// TIA Portal V16 program export: 2 tag tables, 2 data types, 2 data blocks, 72 code blocks (in call order from the OBs), 28 instance data blocks

VAR_GLOBAL   // PLC tag table "Стандартная таблица переменных"
   "K1-112 2L1" AT %I0.0 : Bool;   // Реле безопастности К10 ОСНОВНАЯ напряжение управления
   "K1-113/1 3L1" AT %I0.1 : Bool;   // Реле безопастности К11 концевики группа 211,212,213,214
   "K1-113/2 4L1" AT %I0.2 : Bool;   // Реле безопастности К21 группа 221,222,224,225,231-235,311,312,313-317
   "K1-113/3 5L1" AT %I0.3 : Bool;   // Релле безопасности К31 группа 321,322,324
   "k1-113/4 6L1" AT %I0.4 : Bool;   // Релле безопасности К41 группа 331,332-337
   Varalla AT %I0.5 : Bool;   // резерв
   Varalla1 AT %I0.6 : Bool;   // резерв
   Varalla2 AT %I0.7 : Bool;   // резерв
   "211K1/211K2" AT %I1.0 : Bool;   // М211 включен сигналы
   "212K1" AT %I1.1 : Bool;   // Контактор К1 Включен М212 сигналы
   "213K1" AT %I1.2 : Bool;   // контактор К1 Включен М213 сигналы
   "311K1/311K2" AT %I1.3 : Bool;   // М311 включен сигналы
   Varalla3 AT %I1.4 : Bool;   // резерв
   Varalla4 AT %I1.5 : Bool;   // резерв
   Varalla5 AT %I1.6 : Bool;   // резерв
   Varalla6 AT %I1.7 : Bool;   // резерв
   "221K1" AT %I2.0 : Bool;   // М221 включен сигналы
   "222K1" AT %I2.1 : Bool;   // Контактор К1 Включен М222 сигналы
   "223K1" AT %I2.2 : Bool;   // Обратная связь
   "224K1" AT %I2.3 : Bool;   // М224 включен сигналы
   "225K1" AT %I2.4 : Bool;   // Контактор К1 Включен М225 сигналы
   "330K1" AT %I2.5 : Bool;   // Контактор К1 Включен М330 сигнал
   Varalla8 AT %I2.6 : Bool;   // резерв
   Varalla9 AT %I2.7 : Bool;   // резерв
   "231K1" AT %I3.0 : Bool;   // Контактор К1 Включен М231 сигналы
   "232K1" AT %I3.1 : Bool;   // Контактор К1- Включен М232 сигналы
   "233K1" AT %I3.2 : Bool;   // Контактор К1- Включен М233 сигналы
   "234K1" AT %I3.3 : Bool;   // М234 включен сигналы
   "235K1/235K2" AT %I3.4 : Bool;   // М235 включен сигналы
   Varalla10 AT %I3.5 : Bool;   // резерв
   Varalla11 AT %I3.6 : Bool;   // резерв
   Varalla12 AT %I3.7 : Bool;   // резерв
   "214K1" AT %I4.0 : Bool;   // М214 включен сигналы
   "312K1" AT %I4.1 : Bool;   // М312 включен сигналы
   "313K1/313K2" AT %I4.2 : Bool;   // М313 включен сигналы
   "314K1" AT %I4.3 : Bool;   // М314 включен сигналы
   "315K1" AT %I4.4 : Bool;   // М315 включен сигналы
   "316K1" AT %I4.5 : Bool;   // М316 включен сигналы
   "317K1" AT %I4.6 : Bool;   // Контактор К1 включен М317 сигналы
   Varalla13 AT %I4.7 : Bool;   // резерв
   "321K1/321K2" AT %I5.0 : Bool;   // М321 включен сигналы
   "322K1/322K2" AT %I5.1 : Bool;   // М322 включен сигналы
   "323K1/323K2" AT %I5.2 : Bool;   // М323 включен сигнал
   "K1-324U.1" AT %I5.3 : Bool;   // ПЧТ 324 в работе сигналы
   "325K1" AT %I5.4 : Bool;   // Контактор К1 М325 сигнал
   Varalla15 AT %I5.5 : Bool;   // резерв
   Varalla16 AT %I5.6 : Bool;   // резеов
   Varalla17 AT %I5.7 : Bool;   // резерв
   "331K1" AT %I6.0 : Bool;   // М331 включен сигналы
   "332K1" AT %I6.1 : Bool;   // Контактор К1- включен М332 сигналы
   "333K1" AT %I6.2 : Bool;   // Контактор К1 -включен М333 сигналы
   "334K1" AT %I6.3 : Bool;   // Контактор К1- включен М334 сигналы
   "335K1" AT %I6.4 : Bool;   // Контактор К1- включен М335 сигналы
   "336K1" AT %I6.5 : Bool;   // Контактор К1- включен М336 сигналы
   "337K1" AT %I6.6 : Bool;   // Контактор К1-включен М337 сигнал
   "K1-323U1" AT %I6.7 : Bool;   // ПЧТ 312 в работе сигналы
   "K1-212U1" AT %I7.0 : Bool;   // ПЧТ 212 в работе сигналы
   "K1-213U1" AT %I7.1 : Bool;   // ПЧТ 213 в работе сигналы
   "K1-215U1" AT %I7.2 : Bool;   // ПЧТ 215 в работе сигналы
   "K1-222U1" AT %I7.3 : Bool;   // ПЧТ 222 в работе сигналы
   "K1-225U1" AT %I7.4 : Bool;   // Пчт 225 в работе сигналы
   "K1-231U1" AT %I7.5 : Bool;   // ПЧТ 231 в работе сигналы
   "K1-233U1" AT %I7.6 : Bool;   // ПЧТ 233 в работе сигналы
   "K1-317U1" AT %I7.7 : Bool;   // ПЧТ 317 в работе сигналы
   "K1-332U1" AT %I8.0 : Bool;   // ПЧТ 332 в работе сигналы
   "K1-333U1" AT %I8.1 : Bool;   // ПЧТ 333 в работе сигналы
   "K1-334U1" AT %I8.2 : Bool;   // ПЧТ 334 в работе сигналы
   "K1-335U1" AT %I8.3 : Bool;   // ПЧТ 335 в работе сигналы
   "K1-336U1" AT %I8.4 : Bool;   // ПЧТ 336 в работе сигналы
   "K1-223U1" AT %I8.5 : Bool;   // ПЧТ М223 в работе сигнал
   "K1-324U1" AT %I8.6 : Bool;   // ПЧТ М324 в работе сигнал
   "K1-325U1" AT %I8.7 : Bool;   // ПЧТ М325 в работе сигнал
   "K1/112-S1" AT %I9.0 : Bool;   // Состояние концевика 112S1 сигналы
   "K1/112-S2" AT %I9.1 : Bool;   // Состояние концевика 112S2 сигналы
   "K1/112-S3" AT %I9.2 : Bool;   // Состояние концевика 112S3 сигналы
   Varalla22 AT %I9.3 : Bool;   // резерв
   "K1/113-S11" AT %I9.4 : Bool;   // Состояние концевиков 113S11 сигналы
   "K1/113-S12" AT %I9.5 : Bool;   // Состояние концевиков 113S12 сигналы
   "k1/113-S13" AT %I9.6 : Bool;   // Состояние концевиков 113S13 сигналы
   "FC 323.1" AT %I9.7 : Bool;   // Датчик блокировки поштучной
   "FC 323.2" AT %I10.0 : Bool;   // Датчик на останов основной горки
   "FC 223.1" AT %I10.1 : Bool;   // Начало зоны оценки
   "FC 223.2" AT %I10.2 : Bool;   // Конец зоны оценки
   "FC 223.3" AT %I10.3 : Bool;   // Сброс доски в брак
   FC_323_1 AT %I10.4 : Bool;   // резерв
   Key_Faser AT %I10.5 : Bool;   // индуктивник положения поштучной выдачи
   Varalla30 AT %I10.6 : Bool;   // резерв
   Varalla31 AT %I10.7 : Bool;   // резерв
   "Lift Upp" AT %I11.0 : Bool;   // Лифт вниз
   "Lift Down" AT %I11.1 : Bool;   // Лифт в верх
   "sloi doski" AT %I11.2 : Bool;   // Слой доски 1
   "sloi doski2" AT %I11.3 : Bool;   // Слой доски 2
   "doska v priymke elevator" AT %I11.4 : Bool;   // Доска в приямке элеватора
   koncevik1 AT %I11.5 : Bool;   // концевик 1(середина приемного транспортера)
   koncevik2 AT %I11.6 : Bool;   // концевик 2 (вилы лифта приемного транспортера)
   "nakloniy transporter" AT %I11.7 : Bool;   // наклонный транспортер датчик
   "1,8m" AT %I12.0 : Bool;   // 1,8 длинна
   "2,1m" AT %I12.1 : Bool;   // 2,1 длинна
   "2,4m" AT %I12.2 : Bool;   // 2,4 длинна
   "2,7m" AT %I12.3 : Bool;   // 2,7 длинна
   "3,0m" AT %I12.4 : Bool;   // 3,0 длинна
   "3,3m" AT %I12.5 : Bool;   // 3,3 длинна
   "3,6m" AT %I12.6 : Bool;   // 3,6 длинна
   "3,9m" AT %I12.7 : Bool;   // 3,9 длинна
   "4,2m" AT %I13.0 : Bool;   // 4,2 длинна
   "4,5m" AT %I13.1 : Bool;   // 4,5 длинна
   "4,8m" AT %I13.2 : Bool;   // 4,8 длинна
   "5,1m" AT %I13.3 : Bool;   // 5,1 длинна
   "5,4m" AT %I13.4 : Bool;   // 5,4 длинна
   "5,7m" AT %I13.5 : Bool;   // 5,7 длинна
   "6,0m" AT %I13.6 : Bool;   // 6,0 длинна
   PodBort_1 AT %I13.7 : Bool;   // Положение подвижного борта_1
   PodBort_2 AT %I14.0 : Bool;   // Положение подвижного борта _2
   K312Fault AT %I14.1 : Bool;   // Авария частотника 312
   "S14.2" AT %I14.2 : Bool;   // Максимальная ширина доски концевик М225 зона
   "S14.3" AT %I14.3 : Bool;   // Минимальная ширина доски концевик М225 зона
   "B14.4" AT %I14.4 : Bool;   // счет доски М225 зона после бобышек
   "B14.5" AT %I14.5 : Bool;   // счет доски М225 зона после бобышек
   "K-312U1" AT %I14.6 : Bool;   // ПЧТ 312 В работе
   "S14.7" AT %I14.7 : Bool;   // заднее положение вил
   "S15.0" AT %I15.0 : Bool;   // замедление вил назад
   "S15.1" AT %I15.1 : Bool;   // замедление в перед вил
   "S15.2" AT %I15.2 : Bool;   // Переднее положение вил
   "311_S1" AT %I15.3 : Bool;   // Запрет двиджения М311
   Index AT %I15.4 : Bool;   // Индексная точка энкодера
   "B15.5" AT %I15.5 : Bool;   // вилы в верху
   "311_S2" AT %I15.6 : Bool;   // Ручное управление М311
   "B15.7" AT %I15.7 : Bool;   // вилы в низу
   FC_232_1 AT %I16.0 : Bool;   // набор слоя пакета на лифте1
   "S16.1" AT %I16.1 : Bool;   // лифт ПфМ в низу
   "S16.2" AT %I16.2 : Bool;   // лифт ПФМ в верху
   FC_225_Upor AT %I16.3 : Bool;   // датчик доски на упорах перед транспортером с бобышками
   "E16.4" AT %I16.4 : Bool;   // Уровень Гидростанции Основной
   FC_232_2 AT %I16.5 : Bool;   // Набор слоя пакета на лифте2
   KeyFazerPFM_repeater AT %I16.6 : Bool;   // Второй кейфазер на транспортер бобышек
   KeyFazerPFM AT %I16.7 : Bool;   // кейфазер для транспортера бобышек
   "B17.0" AT %I17.0 : Bool;   // наличие прокладок на М312
   "B17.1" AT %I17.1 : Bool;   // наличие прокладки в М314
   "B17.2" AT %I17.2 : Bool;   // наличие прокладки в М315
   "234.4" AT %I17.3 : Bool;   // второй датчик наличия прокладки перед каруселью
   "234.1" AT %I17.4 : Bool;   // 234.1 прокладка на выдаче(датчик)
   "234.2" AT %I17.5 : Bool;   // 234.2 прокладка максимальный слой
   "234.3" AT %I17.6 : Bool;   // 234.3 перекос прокладки (Авария)
   Fc316 AT %I17.7 : Bool;   // Датчик в конце М316 перед элеватором1
   "B18.0" AT %I18.0 : Bool;   // рейкоукладчик в верху
   "B18.1" AT %I18.1 : Bool;   // второй индуктив на позиционирование карусели
   "S18.2" AT %I18.2 : Bool;   // среднее положение рейкоукладчика
   "S18.3" AT %I18.3 : Bool;   // рейкоукладчик в низу
   "B18.4" AT %I18.4 : Bool;   // датчик положения захвата прокладки открыто
   "B18.5" AT %I18.5 : Bool;   // датчик положени захвата прокладки закрыто
   "B18.6" AT %I18.6 : Bool;   // сигнал набора слоя
   "B18.7" AT %I18.7 : Bool;   // Остановка транспортера прокладок
   "B19.0" AT %I19.0 : Bool;   // Обратный ход транспортера прокладок ДАТЧИК
   Varalla35 AT %I19.1 : Bool;   // резерв
   Varalla36 AT %I19.2 : Bool;   // резерв
   Varalla37 AT %I19.3 : Bool;   // резерв
   Varalla38 AT %I19.4 : Bool;   // резерв
   Varalla39 AT %I19.5 : Bool;   // резерв
   Varalla40 AT %I19.6 : Bool;   // резерв
   Varalla41 AT %I19.7 : Bool;   // резерв
   Varalla42 AT %I20.0 : Bool;   // резерв
   Varalla43 AT %I20.1 : Bool;   // резерв
   Varalla44 AT %I20.2 : Bool;   // резерв
   Varalla45 AT %I20.3 : Bool;   // резерв
   Varalla46 AT %I20.4 : Bool;   // резерв
   Varalla47 AT %I20.5 : Bool;   // резерв
   Varalla48 AT %I20.6 : Bool;   // резерв
   Varalla49 AT %I20.7 : Bool;   // резерв
   Varalla50 AT %I21.0 : Bool;   // резерв
   Varalla51 AT %I21.1 : Bool;   // резерв
   Varalla52 AT %I21.2 : Bool;   // резерв
   Varalla53 AT %I21.3 : Bool;   // резерв
   Varalla54 AT %I21.4 : Bool;   // резерв
   Varalla55 AT %I21.5 : Bool;   // резерв
   Varalla56 AT %I21.6 : Bool;   // резерв
   Varalla57 AT %I21.7 : Bool;   // резерв
   "B22.0" AT %I22.0 : Bool;   // доска в конце роликового транспортера(брак)
   "B22.1" AT %I22.1 : Bool;   // доска в начале роликового транспортера(брак)
   "S22.2" AT %I22.2 : Bool;   // вилы брака ПФМ в перед
   "S22.3" AT %I22.3 : Bool;   // вилы брака ПФМ назад
   "B22.4" AT %I22.4 : Bool;   // лифт брака ПФМ в верху
   "B22.5" AT %I22.5 : Bool;   // лифт брака ПФМ в низу
   "B22.6" AT %I22.6 : Bool;   // Слой на вилах брака ПФМ
   "FC 22.7" AT %I22.7 : Bool;   // Счет доски слоя на пфм Брака
   "B23.0" AT %I23.0 : Bool;   // Пакет на основном разгрузочном транспортере3
   "B23.1" AT %I23.1 : Bool;   // пакет на разгрузочном транспортере 2
   M324Sync AT %I23.2 : Bool;   // индуктив синхронизации М 324
   Varalla60 AT %I23.3 : Bool;   // резерв
   Varalla61 AT %I23.4 : Bool;   // резерв
   Varalla62 AT %I23.5 : Bool;   // резерв
   "FC 23.6" AT %I23.6 : Bool;   // Упоры подняты ПФМ брака
   "FC 23.7" AT %I23.7 : Bool;   // Упоры опущены ПФМ брака
   S76 AT %I24.0 : Bool;   // стоповая кнопка OP1
   "S76.1" AT %I24.1 : Bool;   // Включение напряжения управления
   "S76.2" AT %I24.2 : Bool;   // Подтверждение ошибки
   "S76.3" AT %I24.3 : Bool;   // Гидравлика линии в положении включено
   "E76.4" AT %I24.4 : Bool;   // Старт гидравлики
   "S76.5" AT %I24.5 : Bool;   // авто включение и выключение загрузчика ( режим авто всей загрузки)
   "S76.6" AT %I24.6 : Bool;   // авто М211 приемный транспортер
   "E76.7" AT %I24.7 : Bool;   // вперед М211 приемный транспортер в автомате
   "S77.0" AT %I25.0 : Bool;   // авто М222 горка
   "E77.1" AT %I25.1 : Bool;   // вперед М222 горка в автомате
   "S77.2" AT %I25.2 : Bool;   // Квитирование зоны 1(от горки до ПФМ)
   "S77.3" AT %I25.3 : Bool;   // Квитирование зоны выгрузки
   "S77.4" AT %I25.4 : Bool;   // Квитирование зоны 2 (ПФМ брака)
   "S77.5" AT %I25.5 : Bool;   // авто режим зоны 1( включено, выключено) ( от горки до ПФМ)
   "S77.6" AT %I25.6 : Bool;   // Выдвинуть упоры поштучника
   "E77.7" AT %I25.7 : Bool;   // Убрать упоры поштучника
   "S78.0" AT %I26.0 : Bool;   // Вилы выдвинуть
   "E78.1" AT %I26.1 : Bool;   // Вилы задвинуть
   "S78.2" AT %I26.2 : Bool;   // Вилы опустить
   "E78.3" AT %I26.3 : Bool;   // Вилы поднять
   "S78.4" AT %I26.4 : Bool;   // Лифт опустить
   "E78.5" AT %I26.5 : Bool;   // Лифт поднять
   "S78.6" AT %I26.6 : Bool;   // рейкоукладчик вниз
   "E78.7" AT %I26.7 : Bool;   // рейкоукладчик вверх
   "S79.0" AT %I27.0 : Bool;   // принудительно завершить сборку пакета
   "S79.1" AT %I27.1 : Bool;   // авто подача прокладки(включен,выключен)
   "E79.2" AT %I27.2 : Bool;   // резерв
   "S79.3" AT %I27.3 : Bool;   // авто режим ПФМ брака (включено,выключено)
   "S79.4" AT %I27.4 : Bool;   // Сброс с рольганга(брака) вперпед
   "S79.5" AT %I27.5 : Bool;   // Транспортер набора слоя ( брака) вперед
   "S79.6" AT %I27.6 : Bool;   // вилы( брака) вперед
   "E79.7" AT %I27.7 : Bool;   // вилы( брака) назад
   "S80.0" AT %I28.0 : Bool;   // Упоры слоя ПФМ( брака)
   "E80.1" AT %I28.1 : Bool;   // Упоры слоя ПФМ( брака)
   "S80.2" AT %I28.2 : Bool;   // Лифт ПФМ(брака) опустить
   "E80.3" AT %I28.3 : Bool;   // Лифт ПФМ(брака) поднять
   "S80.4" AT %I28.4 : Bool;   // поднять, опустить Подвижный борт(М235)
   "S80.5" AT %I28.5 : Bool;   // вперед подвижный борт(М235)
   "E80.6" AT %I28.6 : Bool;   // назад подвижный борт(М235)
   "S80.7" AT %I28.7 : Bool;
   Varalla106 AT %I29.0 : Bool;   // резерв
   Varalla107 AT %I29.1 : Bool;   // резерв
   Varalla108 AT %I29.2 : Bool;   // резерв
   Varalla109 AT %I29.3 : Bool;   // резерв
   Varalla110 AT %I29.4 : Bool;   // резерв
   Varalla111 AT %I29.5 : Bool;   // резерв
   Varalla112 AT %I29.6 : Bool;   // резерв
   Varalla113 AT %I29.7 : Bool;   // резерв
   "S82.0" AT %I30.0 : Bool;   // Стоп ОР2
   "S81.1" AT %I30.1 : Bool;   // Приемный транспортер вперед ОР2
   "E82.2" AT %I30.2 : Bool;   // Приемный транспортер назад ОР2
   "S82.3" AT %I30.3 : Bool;   // Авто загрузка включена,выключена ОР2
   "S82.4" AT %I30.4 : Bool;   // Лифт загрузки поднять ОР2
   "E82.5" AT %I30.5 : Bool;   // Лифт загрузки опустить ОР2
   "S82.6" AT %I30.6 : Bool;   // Наклонный транспортер авто ОР2
   "E82.7" AT %I30.7 : Bool;   // Авто наклонный транспортер вперед ОР2
   "S83.0" AT %I31.0 : Bool;   // Ленточный транспортер удаления прокладок назад ОР2
   "E83.1" AT %I31.1 : Bool;   // Ленточный транспортер удаления прокладок вперед ОР2
   "E83.2" AT %I31.2 : Bool;   // Горка прокладок 1 авто ОР2
   "E83.3" AT %I31.3 : Bool;   // Горка прокладок 1 вперед ОР2(авто)
   "S83.4" AT %I31.4 : Bool;   // Квитирование зоны 1 ОР2
   Varalla114 AT %I31.5 : Bool;   // резерв
   Varalla115 AT %I31.6 : Bool;   // резерв
   Varalla116 AT %I31.7 : Bool;   // резерв
   "S84.0" AT %I32.0 : Bool;   // Стоп ОР3
   "S84.1" AT %I32.1 : Bool;   // Транспортер М317 прокладок вперед ОР3
   "E84.2" AT %I32.2 : Bool;   // Транспортер М317 прокладок назад ОР3
   "S84.3" AT %I32.3 : Bool;   // Дозированиe включено ОР3
   "S84.4" AT %I32.4 : Bool;   // авто подача прокладок включена, выключена ОР3
   "S84.5" AT %I32.5 : Bool;   // Рейкоукладчик вниз ОР3
   "E84.6" AT %I32.6 : Bool;   // Рейкоукладчик вверх ОР3
   "S84.7" AT %I32.7 : Bool;   // Открыть стакан прокладки ОР3
   "E85.0" AT %I33.0 : Bool;   // Закрыть стакан прокладки ОР3
   "S85.1" AT %I33.1 : Bool;
   "E85.2" AT %I33.2 : Bool;
   "S85.3" AT %I33.3 : Bool;   // авто горка прокладок 2,3 ОР3
   "E85.4" AT %I33.4 : Bool;   // горка 2,3 прокладок вперед(авто) ОР3
   "S85.5" AT %I33.5 : Bool;   // М234 назад ОР3
   "E85.6" AT %I33.6 : Bool;   // М234 вперед транспортер прокладок перед крючками ОР3
   "S85.7" AT %I33.7 : Bool;   // Квитирование зоны прокладок ОР3
   "S86.0" AT %I34.0 : Bool;   // Лифт ПФМ вниз ОР3
   "E86.1" AT %I34.1 : Bool;   // ЛИфт ПФМ вверх ОР3
   "S86.2" AT %I34.2 : Bool;   // Ролики лифта ПФМ вперед ОР3
   "S86.3" AT %I34.3 : Bool;   // ПФМ Основное Авто включено, выключено ОР3
   "S86.4" AT %I34.4 : Bool;   // Подтверждение неисправности ОР3
   "S86.5" AT %I34.5 : Bool;   // датчик
   Varalla117 AT %I34.6 : Bool;   // резерв
   Varalla118 AT %I34.7 : Bool;   // резерв
   "S87.0" AT %I35.0 : Bool;   // Кнопка брака ОР1.1
   "S87.1" AT %I35.1 : Bool;   // Горка авто ОР1.1
   "E87.2" AT %I35.2 : Bool;   // Горка ОР1.1 (авто)
   "S87.3" AT %I35.3 : Bool;   // датчик перекоса перед плавниками
   "S87.4" AT %I35.4 : Bool;   // набор ковра перед плавниками
   Varalla119 AT %I35.5 : Bool;   // резерв
   Varalla120 AT %I35.6 : Bool;   // резерв
   Varalla121 AT %I35.7 : Bool;   // резерв
   "S88.0" AT %I36.0 : Bool;   // Стоп ОР4
   "K3.3" AT %I36.1 : Bool;   // работа подвижного борта ОР4
   "S88.2" AT %I36.2 : Bool;   // Выкатной транспортер 1 ПФМ назад ОР4
   "E88.3" AT %I36.3 : Bool;   // Выкатной транспортер 1 ПФМ вперед ОР4
   "S88.4" AT %I36.4 : Bool;   // Выкатной транспортер 2 ПФМ назад ОР4
   "S88.5" AT %I36.5 : Bool;   // Выкатной транспортер 2 ПФМ вперед ОР4
   "E88.6" AT %I36.6 : Bool;   // резерв ОР4
   "S88.7" AT %I36.7 : Bool;   // резерв ОР4
   "S89.0" AT %I37.0 : Bool;   // Выкатной транспортер 3 ПФМ назад ОР4
   "S89.1" AT %I37.1 : Bool;   // Выкатной транспортер 3 ПФМ вперед ОР4
   "S89.2" AT %I37.2 : Bool;   // Квитирование ОР4
   "S89.3" AT %I37.3 : Bool;   // датчик ОР4
   Varalla122 AT %I37.4 : Bool;   // резерв ОР4
   Varalla123 AT %I37.5 : Bool;   // резерв ОР4
   Varalla124 AT %I37.6 : Bool;   // резерв ОР4
   Varalla125 AT %I37.7 : Bool;   // резерв ОР4
   "S90.0" AT %I38.0 : Bool;   // Стоп ОР5
   "S90.1" AT %I38.1 : Bool;   // М331 вперед ленточный транспортер брака ОР5
   "S90.2" AT %I38.2 : Bool;   // М332 вперед сбрасыватель рольганга брака ОР5
   Varalla126 AT %I38.3 : Bool;   // резерв
   "S90.4" AT %I38.4 : Bool;   // Вилы ПФМ брака назад ОР5
   "E90.5" AT %I38.5 : Bool;   // Вилы ПФМ брака вперед ОР5
   "S90.6" AT %I38.6 : Bool;   // Опустить упоры формирования слоя на ПФМ брака ОР5
   "E90.7" AT %I38.7 : Bool;   // Поднять упоры формирования слоя на ПФМ брака ОР5
   "S91.0" AT %I39.0 : Bool;   // Лифт брака ПФМ опустить ОР5
   "E91.1" AT %I39.1 : Bool;   // Лифт брака ПФМ поднять ОР5
   "S91.2" AT %I39.2 : Bool;   // квитирование ПФМ 2
   Varalla127 AT %I39.3 : Bool;   // резерв
   Varalla128 AT %I39.4 : Bool;   // резерв
   Varalla129 AT %I39.5 : Bool;   // резерв
   Varalla130 AT %I39.6 : Bool;   // резерв
   Varalla131 AT %I39.7 : Bool;   // резерв
   "K1-212U" AT %QW512 : Int;
   "K1-213U" AT %QW514 : Int;
   "K1-215U" AT %QW516 : Int;
   "K1-222U" AT %QW518 : Int;
   "K1-225U" AT %QW520 : Int;
   "K1-231U" AT %QW522 : Int;
   "K1-233U" AT %QW524 : Int;
   "K1-317U" AT %QW526 : Int;
   "K1-332U" AT %QW528 : Int;
   "K1-333U" AT %QW530 : Int;
   "K1-334U" AT %QW532 : Int;
   "K1-335U" AT %QW534 : Int;
   "K1-336U" AT %QW536 : Int;
   "K1-223U" AT %QW538 : Int;
   "k1-323U" AT %QW540 : Int;
   "K1-325U" AT %QW542 : Int;
   "K1-112x1" AT %Q0.0 : Bool;   // релле Сирены
   "Sk1-113" AT %Q0.1 : Bool;   // разрешение на запуск релле К10 безопастность
   "K1-113X1" AT %Q0.2 : Bool;   // разрешение на запуск релле К11 безопастность
   "K1-113X2" AT %Q0.3 : Bool;   // разрешение на запуск релле К21 безопастность
   "K1-113X3" AT %Q0.4 : Bool;   // разрешение на запуск релле К31 безопастность
   "K1-113X4" AT %Q0.5 : Bool;   // разрешение на запуск релле К41 безопастность
   Varalla65 AT %Q0.6 : Bool;   // резерв
   Varalla66 AT %Q0.7 : Bool;   // резерв
   "K1-211X1" AT %Q1.0 : Bool;   // М211 вперед загрузочный транспортер
   "K1-211X1.1" AT %Q1.1 : Bool;   // М211 назад загрузочный транспортер
   "K1-212X1" AT %Q1.2 : Bool;   // контактор К1-212 ПЧТ запуск лифт
   "K1-212X1.1" AT %Q1.3 : Bool;   // Растормаживание М212 лифт
   "K1-213X1" AT %Q1.4 : Bool;   // контактор К1-213 ПЧТ запуск наклонный транспортер
   "K1-311X1" AT %Q1.5 : Bool;   // запуск ленточного транспортера удалителя прокладок M311
   Varalla68 AT %Q1.6 : Bool;   // резерв
   Varralla69 AT %Q1.7 : Bool;   // резерв
   "K1-221X1" AT %Q2.0 : Bool;   // запуск М221 гидростанция1
   "K1-222X1" AT %Q2.1 : Bool;   // Запуск контактора К1-222 ПЧТ основной элеватор
   "K1-223X1" AT %Q2.2 : Bool;   // запуск М223 Цепной после поштучника
   "K1-224X1" AT %Q2.3 : Bool;   // запуск М224 выдвинуть упоры поштучника
   "K1-224-x1.1" AT %Q2.4 : Bool;   // запуск М224 задвинуть упоры поштучника
   "K1-225X1" AT %Q2.5 : Bool;   // включение контактора К1-225 ПЧТ транспортер бобышек
   "K1-231X1" AT %Q2.6 : Bool;   // включение контактора К1-231 ПЧТ ролики торцовочные
   "K1-232X1" AT %Q2.7 : Bool;   // включение контактора К1-232 ПЧТ Лифт ПФМ
   "K1-232X1.1" AT %Q3.0 : Bool;   // Тормоз Лифта ПФМ
   "K1-233X1" AT %Q3.1 : Bool;   // включение контактора К1-233 ПЧТ вилы ПФМ
   "K1-234X1" AT %Q3.2 : Bool;   // запуск М234 транспортер прокладок перед крючками ПФМ
   "K1-235X1" AT %Q3.3 : Bool;   // запуск М235 вперед подвижный борт
   "K1-214X1" AT %Q3.4 : Bool;   // запуск М214 транспортер загрузки прокладок
   "K1-330X1" AT %Q3.5 : Bool;   // запуск М330 контактора лента брака2
   "K1-312X1" AT %Q3.6 : Bool;   // запуск М312 первая горка прокладок
   "K1-313X1" AT %Q3.7 : Bool;   // запуск М313 вперед транспортер прокладок после первой горки
   "K1-313X1.1" AT %Q4.0 : Bool;   // запуск М313 назад транспортера прокладок после первой горки
   "K1-314X1" AT %Q4.1 : Bool;   // запуск М314 горка прокладок 2
   "K1-315X1" AT %Q4.2 : Bool;   // запуск М315 горка прокладок 3
   "K1-316X1" AT %Q4.3 : Bool;   // запуск М316 транспортер загрузки прокладок в горку 2
   "K1-317X1" AT %Q4.4 : Bool;   // включение контактора К1-317 ПЧТ основной транспортер прокладок
   "K1-317X1.1" AT %Q4.5 : Bool;   // тормоз М317
   "K1-321X1" AT %Q4.6 : Bool;   // запуск М321 вперед выкатной транспортер ПФМ
   "K1-321X1.1" AT %Q4.7 : Bool;   // запуск М321 назад выкатной транспортер ПФМ
   "K1-322X1" AT %Q5.0 : Bool;   // запуск М322 вперед выкатной транспортер ПФМ2
   "K1-322X1.1" AT %Q5.1 : Bool;   // Запуск М322 назад выкатной транспортер ПФМ2
   "K1-323X1" AT %Q5.2 : Bool;   // Запуск контактора М323 маленький после элеватора
   "K1-325U2" AT %Q5.3 : Bool;   // Старт ПЧТ М325 набор слоя основной
   "K1-324U2" AT %Q5.4 : Bool;   // команда на ПЧТ вперед М324 выгрузка покета выкатной ПФМ3
   "K1-324U2.2" AT %Q5.5 : Bool;   // команда на ПЧТ назад М324 выгрузка покета выкатной ПФМ3
   "K1-325X1" AT %Q5.6 : Bool;   // Включение контактора К1-325 ПЧТ набор слоя основной
   "K1-235X1.1" AT %Q5.7 : Bool;   // запуск М235 назад подвижный борт
   "K1-331X1" AT %Q6.0 : Bool;   // запуск М331 ленточный транспортер брака
   "K1-332x1" AT %Q6.1 : Bool;   // включение контактора К1-332 ПЧТ сбрасыватель с рольганга (брак)
   "K1--333X1" AT %Q6.2 : Bool;   // включение контактора К1-333 ПЧТ рольганг (брака)
   "K1-334X1" AT %Q6.3 : Bool;   // включение контактора К1-334 ПЧТ транспортер сбора слоя ПФМ брака
   "K1-335X1" AT %Q6.4 : Bool;   // включение контактора К1-335 ПЧТ вилы ПФМ брака
   "K1-336X1" AT %Q6.5 : Bool;   // Включение контактора К1-336 ПЧТ лифт ПФМ брака
   "K1-336X1.1" AT %Q6.6 : Bool;   // Тормоз М336 лифта ПФМ брака
   "K1-337K1" AT %Q6.7 : Bool;   // Контактор пуска Гирдростанции ПФМ Брака
   Varalla70 AT %Q7.0 : Bool;   // резерв
   "K1-312U2" AT %Q7.1 : Bool;   // Старт ПЧТ 312
   Varalla72 AT %Q7.2 : Bool;   // резерв
   Varalla73 AT %Q7.3 : Bool;   // резерв
   Varalla74 AT %Q7.4 : Bool;   // резерв
   Varalla75 AT %Q7.5 : Bool;   // резерв
   Varalla76 AT %Q7.6 : Bool;   // резерв
   Varalla77 AT %Q7.7 : Bool;   // резерв
   "K1-212U2" AT %Q8.0 : Bool;   // старт ПЧТ М212
   "K1-212U2.2" AT %Q8.1 : Bool;   // Реверс ПЧТ М212
   "K1-213U2" AT %Q8.2 : Bool;   // Старт ПЧТ М213
   "K1-215U2" AT %Q8.3 : Bool;   // Старт ПЧТ 232
   "K1-215U2.2" AT %Q8.4 : Bool;   // Реверс ПЧТ 232
   "K1-222U2" AT %Q8.5 : Bool;   // Старт ПЧТ 222
   "K1-225U2" AT %Q8.6 : Bool;   // Старт ПЧТ 225
   "K1-231U2" AT %Q8.7 : Bool;   // Старт ПЧТ 231
   "K1-233U2" AT %Q9.0 : Bool;   // Старт ПЧТ 233
   "K1-233U2.2" AT %Q9.1 : Bool;   // Реверс ПЧТ 233
   "K1-223U2" AT %Q9.2 : Bool;   // Старт ПЧТ 223
   "K1-332U2" AT %Q9.3 : Bool;   // Старт ПЧТ 332
   "K1-333U2" AT %Q9.4 : Bool;   // Старт ПЧТ 333
   "K1-334U2" AT %Q9.5 : Bool;   // Старт ПЧТ 334
   "K1-335U2" AT %Q9.6 : Bool;   // Старт ПЧТ 335
   "K1-335U2.2" AT %Q9.7 : Bool;   // Реверс ПЧТ 335
   "K1-336U2" AT %Q10.0 : Bool;   // Стасрт ПЧТ 336
   "K1-336U2.2" AT %Q10.1 : Bool;   // Реверс ПЧТ 336
   "K1-317U2" AT %Q10.2 : Bool;   // Старт ПЧТ 317
   "K1-317U2.2" AT %Q10.3 : Bool;   // Реверс ПЧТ 317
   Y223_1 AT %Q12.0 : Bool;   // переворот доски вверх
   Y223_2 AT %Q12.1 : Bool;   // переворот доски вниз
   Y223_3 AT %Q12.2 : Bool;   // сброс в брак вниз
   Y223_4 AT %Q12.3 : Bool;   // сброс в брак вверх
   Y323_1 AT %Q12.4 : Bool;   // упоры перед поштучкой вверх
   Y323_2 AT %Q12.5 : Bool;   // упоры перед поштучкой вниз
   Upor_brak_up AT %Q12.6 : Bool;   // упоры ПФМ брака вверх
   Upor_brak_down AT %Q12.7 : Bool;   // упоры ПФМ брака вниз
   "Y223.3" AT %Q13.0 : Bool;   // перепускной клапан маленькая гидростанция
   "Y223.4" AT %Q13.1 : Bool;   // перепускной клапан маленькая гидростанция
   Varalla89 AT %Q11.6 : Bool;   // резерв
   Varalla90 AT %Q11.7 : Bool;   // резерв
   "K1-323U2" AT %Q10.4 : Bool;   // Старт ПЧТ 323
   "Y12.1" AT %Q10.5 : Bool;   // резерв
   Varalla91 AT %Q10.6 : Bool;   // резерв
   Varalla92 AT %Q10.7 : Bool;   // резерв
   Varalla93 AT %Q11.0 : Bool;   // резерв
   Varalla94 AT %Q11.1 : Bool;   // резерв
   Varalla95 AT %Q11.2 : Bool;   // резерв
   Varalla96 AT %Q11.3 : Bool;   // резерв
   "Y13.0" AT %Q11.4 : Bool;
   "Y13.1" AT %Q11.5 : Bool;
   "Y13.2" AT %Q13.2 : Bool;
   "Y13.3" AT %Q13.3 : Bool;
   "Y13.4" AT %Q13.4 : Bool;
   "Y13.5" AT %Q13.5 : Bool;
   "Y13.6" AT %Q13.6 : Bool;
   "Y13.7" AT %Q13.7 : Bool;
   Line1_1 AT %Q14.0 : Bool;   // вилы вниз
   Line1_2 AT %Q14.1 : Bool;   // вилы вверх
   Line2_1 AT %Q14.2 : Bool;   // упоры перед поштучкой вверх
   Line2_2 AT %Q14.3 : Bool;   // упоры перед поштучкой вниз
   Line3_1 AT %Q14.4 : Bool;   // подвижный борт опустить
   Line3_2 AT %Q14.5 : Bool;   // подвижный борт поднять
   Line4_1 AT %Q14.6 : Bool;   // выдача прокладки вниз
   Line4_2 AT %Q14.7 : Bool;   // выдача прокладки вверх
   Perepusk AT %Q15.0 : Bool;   // перепускной клапан большая гидростанция
   Line5_1 AT %Q15.1 : Bool;   // каретка прокладки вниз
   Line5_2 AT %Q15.2 : Bool;   // каретка прокладки вверх
   Line6_1 AT %Q15.3 : Bool;   // ложементы закрыть
   Line6_2 AT %Q15.4 : Bool;   // ложементы открыть
   Varalla100 AT %Q15.5 : Bool;   // резерв
   Varalla101 AT %Q15.6 : Bool;   // резерв
   Varalla102 AT %Q15.7 : Bool;   // резерв
   "H76.0" AT %Q16.0 : Bool;   // Напряжение управления включено (лампочка) ОР1
   "H76.1" AT %Q16.1 : Bool;   // потверждение аварии (лампочка) ОР1
   "H76.2" AT %Q16.2 : Bool;   // Гидравлика линии в положении включено (лампочка) ОР1
   "H76.3" AT %Q16.3 : Bool;   // авто включение и выключение загрузчика ( режим авто всей загрузки) (лампочка)ОР1
   "H76.4" AT %Q16.4 : Bool;   // разгрусчик открыт (лапмочка) ОР1
   "H76.5" AT %Q16.5 : Bool;   // Квитирование ПФМ 1 (лапмочка)ОР1
   "H76.6" AT %Q16.6 : Bool;   // Квитирование (лампочка)ОР1
   "H76.7" AT %Q16.7 : Bool;   // Квитирование ПФМ 2 (лампочка)ОР1
   "H77.0" AT %Q17.0 : Bool;   // ПФМ 1 авто включено ( лампочка)ОР1
   "H77.1" AT %Q17.1 : Bool;   // авто подача прокладки(включен,выключен) (лампочка)ОР1
   "H77.2" AT %Q17.2 : Bool;   // Авто ПФМ 2 включен (лампочка)ОР1
   Varalla132 AT %Q17.3 : Bool;   // резерв ОР1
   Varalla133 AT %Q17.4 : Bool;   // резерв ОР1
   Varalla134 AT %Q17.5 : Bool;   // резерв ОР1
   Varalla135 AT %Q17.6 : Bool;   // резерв ОР1
   Varalla136 AT %Q17.7 : Bool;   // резерв ОР1
   "H78.0" AT %Q18.0 : Bool;   // Авто загрузка включена,выключена ОР2 (лампочка)
   "H78.1" AT %Q18.1 : Bool;   // квитирование загрузки (лампочка)ОР2
   Varalla137 AT %Q18.2 : Bool;   // резерв
   Varalla138 AT %Q18.3 : Bool;   // резерв
   "A78.4" AT %Q18.4 : Bool;   // Авто подачи прокладок включен (лампочка)ОР3
   "A78.5" AT %Q18.5 : Bool;   // Квитирование прокладок (лампочка)ОР3
   "A78.6" AT %Q18.6 : Bool;   // Авто ПФМ 1 включен ( лампочка) ОР3
   "H78.7" AT %Q18.7 : Bool;   // Авария (лампочка)ОР3
   "H79.0" AT %Q19.0 : Bool;   // Квитирование выгрузки (лампочка) ОР4
   Pakkauspuristin AT %Q19.1 : Bool;
   "A79.2" AT %Q19.2 : Bool;   // резерв
   "A79.3" AT %Q19.3 : Bool;   // резерв
   "H79.4" AT %Q19.4 : Bool;   // Квитирование ПФМ2 (лампочка)
   Varalla139 AT %Q19.5 : Bool;   // резерв
   Varalla140 AT %Q19.6 : Bool;   // резерв
   Varalla141 AT %Q19.7 : Bool;   // резерв
   Lift AT %M20.0 : Bool;
   FALSE AT %M20.1 : Bool;
   M212StartDelay AT %T1 : Timer;   // Задержка перд стартом загрузки пакета на лифт
   Tag_2 AT %T2 : Timer;
   M212DownDelay AT %T3 : Timer;   // Задержка на опускания лифта вниз
   DropDelay AT %T4 : Timer;   // задержка на срабатывания датчиков сброся слоя
   m212waitAfterDrop AT %T6 : Timer;   // Задержка на сброс доски после сброса
   m213DropDelay AT %T7 : Timer;
   M212waitEmptyHole AT %T8 : Timer;   // Ожидание освобождения приямка горки загрузки
   Tag_9 AT %T9 : Timer;
   M211startDelay AT %T10 : Timer;   // задержка старта транспортера при установке пакета погрузчиком
   Tag_11 AT %T11 : Timer;
   Tag_12 AT %T12 : Timer;
   Tag_13 AT %T13 : Timer;
   Tag_14 AT %T14 : Timer;
   Tag_15 AT %T15 : Timer;
   Tag_16 AT %T16 : Timer;
   Tag_17 AT %T17 : Timer;
   Tag_18 AT %T18 : Timer;
   Tag_5 AT %M0.0 : Bool;
   Tag_61 AT %M0.1 : Bool;
   Tag_62 AT %T19 : Timer;
   NaprUpr AT %M0.6 : Bool;   // меркер напряжения управления
   Tag_19 AT %C1 : Counter;
   Tag_20 AT %C2 : Counter;
   HodVil2 AT %M1.2 : Bool;
   Tag_71 AT %T5 : Timer;
   Tag_72 AT %T20 : Timer;
   Tag_73 AT %C3 : Counter;
   Fouls AT %M4.0 : Bool;
   TRUE AT %M4.1 : Bool;
   "Tag_19(1)" AT %T21 : Timer;
   M213AlarmFilter AT %T22 : Timer;
   M214AlarmFilter AT %T23 : Timer;
   "221StartDelay" AT %T24 : Timer;
   "222AlarmFilter" AT %T25 : Timer;
   "223AlarmFilter" AT %T26 : Timer;
   "332AlarmFilter" AT %T27 : Timer;
   "333AlarmFilter" AT %T28 : Timer;
   "334AlarmFilter" AT %T29 : Timer;
   "336DownDelay" AT %T30 : Timer;
   "336AlarmFilter" AT %T31 : Timer;
   "321AlarmFilter" AT %T32 : Timer;
   "322AlarmFilter" AT %T33 : Timer;
   "324AlarmFilter" AT %T34 : Timer;
   "214AlarmFiltr" AT %T35 : Timer;
   "312AlarmFiltr" AT %T36 : Timer;
   "313AlarmFilter" AT %T37 : Timer;
   "316AlarmFiltr" AT %T38 : Timer;
   "314AlarmFilter" AT %T39 : Timer;
   "234AlarmFilter" AT %T40 : Timer;
   Tag_3 AT %M4.7 : Bool;
   "224AlarmFilter" AT %T41 : Timer;
   "225AlarmFilter" AT %T42 : Timer;
   "231AlarmFilter" AT %T43 : Timer;
   "235AlarmFilter" AT %T44 : Timer;
   "311AlarmFilter" AT %T45 : Timer;
   "335AlarmFilter" AT %T46 : Timer;
   "331AlarmFilter" AT %T47 : Timer;
   "233AlarmFilter" AT %T48 : Timer;
   "337AlarmFilter" AT %T49 : Timer;
   "232AlarmFilter" AT %T50 : Timer;
   alarm AT %M2.0 : Bool;
   M323_HoldRun AT %T51 : Timer;
   Tag_1 AT %C4 : Counter;
   Tag_4 AT %T52 : Timer;
   Tag_6 AT %M2.1 : Bool;
   M323_RunTask AT %T53 : Timer;
   Tag_7 AT %T54 : Timer;
   Tag_8 AT %T55 : Timer;
   ElevatorPFM_Defective_cmd_lowering AT %M4.5 : Bool;
   Tag_21 AT %T56 : Timer;
   Tag_22 AT %M40.0 : Bool;
   Tag_23 AT %M40.1 : Bool;
   Tag_24 AT %M40.2 : Bool;
   Tag_25 AT %M40.3 : Bool;
   Tag_26 AT %M40.4 : Bool;
   Tag_27 AT %M40.5 : Bool;
   Tag_28 AT %M40.6 : Bool;
   Tag_29 AT %M40.7 : Bool;
   Tag_30 AT %M41.0 : Bool;
   Tag_31 AT %M41.1 : Bool;
   Tag_32 AT %IW544 : Word;
   Tag_33 AT %IW545 : Word;
   Tag_34 AT %M5.0 : Bool;
   Tag_35 AT %T79 : Timer;
   Tag_36 AT %T78 : Timer;
   Tag_37 AT %T80 : Timer;
   Tag_38 AT %T67 : Timer;
   Tag_39 AT %T68 : Timer;
   Tag_40 AT %T81 : Timer;
   Tag_41 AT %M5.2 : Bool;
   Tag_42 AT %T82 : Timer;
   Tag_43 AT %M5.6 : Bool;
   Tag_44 AT %T83 : Timer;
   Tag_45 AT %M5.7 : Bool;
   Tag_46 AT %T84 : Timer;
   Hill_endTask AT %T85 : Timer;
   Tag_48 AT %M6.0 : Bool;
   Tag_49 AT %M6.1 : Bool;
   Tag_50 AT %M6.2 : Bool;
   Tag_51 AT %T86 : Timer;
   Tag_52 AT %M6.3 : Bool;
   Tag_53 AT %T87 : Timer;
   Tag_54 AT %M41.2 : Bool;
   Tag_55 AT %T88 : Timer;
   Tag_56 AT %T89 : Timer;
   Tag_57 AT %M7.4 : Bool;
   Tag_58 AT %T90 : Timer;
   Tag_59 AT %T92 : Timer;
   Tag_60 AT %M7.2 : Bool;
   Tag_63 AT %T91 : Timer;
   Tag_64 AT %M4.2 : Bool;
   Tag_65 AT %M4.3 : Bool;
   Tag_66 AT %M4.4 : Bool;
   Tag_67 AT %M4.6 : Bool;
   Feed_cmd AT %M5.1 : Bool;
   Tag_69 AT %T93 : Timer;
   Tag_70 AT %M5.3 : Bool;
   Tag_74 AT %T94 : Timer;
   Tag_75 AT %M5.4 : Bool;
   Tag_76 AT %T95 : Timer;
   Tag_77 AT %IW19 : Word;
   Tag_78 AT %IB19 : Byte;
   Tag_79 AT %T96 : Timer;
   EvevatorPFM_Defective_cmd_UP AT %M41.3 : Bool;
   Tag_81 AT %T97 : Timer;
   Tag_82 AT %T98 : Timer;
   Tag_83 AT %T99 : Timer;
   Tag_84 AT %M41.4 : Bool;
   Tag_85 AT %M41.5 : Bool;
   Tag_86 AT %C5 : Counter;
   Tag_87 AT %C6 : Counter;
   StartMakeGasketLayer AT %M41.6 : Bool;
   ElevatorPFM_Defective_cmd_pushPack AT %M41.7 : Bool;
   LayerGetRidOff_flag AT %M42.0 : Bool;
   UporDispenser_permission AT %M42.1 : Bool;
   Tag_92 AT %M42.2 : Bool;
   Tag_93 AT %M42.3 : Bool;
   Tag_94 AT %T100 : Timer;
   Tag_95 AT %T101 : Timer;
   Tag_96 AT %T102 : Timer;
   Tag_97 AT %T103 : Timer;
   Tag_98 AT %T104 : Timer;
   Tag_99 AT %T105 : Timer;
   LampOp3On_Hz AT %M42.4 : Bool;
   Tag_101 AT %T106 : Timer;
   Tag_102 AT %T107 : Timer;
   LampOp3On_NoHz AT %M42.5 : Bool;
   Tag_104 AT %T108 : Timer;
   Tag_105 AT %T109 : Timer;
   Tag_106 AT %T110 : Timer;
   Tag_107 AT %T120 : Timer;
   Tag_108 AT %M10.0 : Bool;
   Tag_109 AT %T121 : Timer;
   Tag_110 AT %M10.1 : Bool;
   Tag_111 AT %T122 : Timer;
   Tag_112 AT %M10.2 : Bool;
   Tag_113 AT %T124 : Timer;
   Tag_114 AT %T111 : Timer;
   SensLineAlarms AT %M42.6 : Bool;
   CarouselManAlarms AT %M10.5 : Bool;
   UporDispenser_down AT %M42.7 : Bool;
   AlarmInfoOnly AT %M43.0 : Bool;
   FC_323_1_delayed AT %T130 : Timer;
   SensorLineRawData AT %IW12 : Word;
   "2Hz" AT %M43.1 : Bool;
   Tag_123 AT %T112 : Timer;
   Tag_124 AT %M43.2 : Bool;
   Tag_125 AT %T113 : Timer;
   Tag_126 AT %T114 : Timer;
   DelayDovodPFM AT %T115 : Timer;
   DelayStartM225 AT %T116 : Timer;
   DelayUporBrak_OFF AT %T117 : Timer;
   FC_323_1_holded AT %T118 : Timer;
   M_334_permission AT %T119 : Timer;
   BoardKickDefect_task AT %T123 : Timer;
   RunM330_M331 AT %T125 : Timer;
   RunM333 AT %T126 : Timer;
END_VAR

VAR_GLOBAL   // PLC tag table "Таблица переменных из SDF_1"
END_VAR

TYPE "PlankOnChain"
// stored: IsFailsafeCompliant false
   STRUCT
      Chain : Bool;   // Цепь, на которйо ледит доска (0 - низкая, 1 - высокая)
      NoEmpty : Bool;   // есть доска на цепи
      Length : Int;   // Длина уложенной доски
   END_STRUCT;
END_TYPE

TYPE "ServIM"
// stored: IsFailsafeCompliant false
   STRUCT
      BtnDU : Bool;   // Включить дистанционный режим
      BtnAU : Bool;   // Отключить дистанционный режим
      BtnFwd : Bool;   // Включить вперёд / выдвинуть
      BtnBwd : Bool;   // Включить назад / задвинуть
      BtnCmdStop : Bool;   // Остановить
      SetSpeedDU : Real;   // Задание на частотник в ДУ
      PrmBtnDU_ON : Bool;   // Разрешение на включение дистанционного режима
      PrmBtnDU_OF : Bool;   // Разрешение на отключение дистанционного режима
      PRMbtn_Back_ON : Bool;   // Разрешение кнопки включения заднего хода
      PRMbtn_Back_OFF : Bool;   // Разрешение кнопки отключения заднего хода
      PrmBtnCmdStop : Bool;   // Разрешение на остановку
      Ready : Bool;   // Готовность к работе
      ON : Bool;   // В работе
      OFF : Bool;   // Не в работе (закрыто)
      Fault : Bool;   // Обобщенная неисправность
      Alarm : Bool;   // Авария
      AU : Bool;   // Автоматическое управление
      MU : Bool;   // Местное управление
      DU : Bool;   // Дистанционный режим включен
      CMD_ON : Bool;   // Запустить ON
      CMD_OFF : Bool;   // Запустить OFF
      BACK : Bool;   // Реверс (задний ход)
      SetSpeed : Real;   // Задание на частотник
   END_STRUCT;
END_TYPE

DATA_BLOCK "ALG"   // DB9
VERSION : 0.1
// stored: AutoNumber true, IsOnlyStoredInLoadMemory false, IsWriteProtectedInAS false
   VAR RETAIN
      Ready_defect : Bool;
      Alarm_defect : Bool;
      Auto_defect : Bool;
      Ready_loading : Bool;
      Alarm_loading : Bool;
      Auto_loading : Bool;
      Ready_Sorting : Bool;
      Alarm_Sorting : Bool;
      Auto_Sorting : Bool;
      Ready_Gasket : Bool;
      Alarm_Gasket : Bool;
      Auto_Gasket : Bool;
      Ready_Rout : Bool;
      Alarm_Rout : Bool;
      Auto_Rout : Bool;
      Reset : Bool;
      start_encoder : Bool := true;   // начать счет энкодера
      reset_encoder : Bool;   // направление влево
      ForceFinishMainPFM : Bool;
      ForceFinishPFMDefect : Bool;
      DefectivePacketIsPushed : Bool;
      PacketReadyRollOut : Bool;   // пакет готов к отгрузке
      EmptyLodems : Bool;
      AddGasketLayer : Bool;   // добавить слой прокладок
      ConfirmGasketsBrak : Bool;   // бит подтверждения на слой брака
      ModeChang : Bool;
      STOP : Bool;   // глобальный тсоп
      VirtualAuto : Bool;
      RampSyncSig : Bool;
      HELPER : Bool;
      TestCounter : Int;
      TestCounter2 : Int;
      LayerVolume : DInt;   // текущий объем пакета
      Volume : DInt;
      Meandr : Int;   // счет для меандра
      PermMovM323 : Time;   // тайминг на работу упоров
      SqueezeRamp : Time := T#1ms;   // задержка на движение рамы
      SqueezeUporPFM : Time;
   END_VAR
BEGIN
END_DATA_BLOCK

DATA_BLOCK "VELOCITY"   // DB19
VERSION : 0.1
// stored: AutoNumber true, IsOnlyStoredInLoadMemory false, IsWriteProtectedInAS false
   VAR RETAIN
      GeneralSpeed : Real;   // Общая скорость линии
      koef_M_332 : Real := 0.4;   // сброс с рольганга
      koef_M_333 : Real := 0.24;   // рольганг брака
      koef_M_334 : Real := 0.2;   // набор слоя
      koef_M_335 : Real := 0.12;   // вилы
      koef_M_336 : Real := 0.2;   // лифт
      koef_M_212 : Real := 0.2;   // лифт загрузки
      koef_M_213 : Real := 0.45;   // наклонный транспортер
      koef_M_222 : Real := 0.09;   // главная горка
      koef_M_231 : Real := 0.12;   // Ролики прибортовщики
      koef_M_325 : Real := 0.7;   // Довод слоя
      koef_M_225 : Real := 0.142;   // Транспортер с бобышками
      koef_M_223 : Real := 0.3;   // зона оценки
      koef_M_232 : Real := 0.25;   // лифт ПФМ
   END_VAR
BEGIN
END_DATA_BLOCK

ORGANIZATION_BLOCK "Main"   // OB1, LAD, ProgramCycle
TITLE = "Main Program Sweep (Cycle)"
VERSION : 0.1
// stored: IsIECCheckEnabled false
   VAR_TEMP
      OB1_EV_CLASS : Byte;   // Bits 0-3 = 1 (Coming event), Bits 4-7 = 1 (Event class 1)
      OB1_SCAN_1 : Byte;   // 1 (Cold restart scan 1 of OB 1), 3 (Scan 2-n of OB 1)
      OB1_PRIORITY : Byte;   // Priority of OB Execution
      OB1_OB_NUMBR : Byte;   // 1 (Organization block 1, OB1)
      OB1_RESERVED_1 : Byte;   // Reserved for system
      OB1_RESERVED_2 : Byte;   // Reserved for system
      BoardPosition : Int;   // Позиция подвижного борта
      OB1_PREV_CYCLE : Int;   // Cycle time of previous OB1 scan (milliseconds)
      OB1_MIN_CYCLE : Int;   // Minimum cycle time of OB1 (milliseconds)
      OB1_MAX_CYCLE : Int;   // Maximum cycle time of OB1 (milliseconds)
      OB1_DATE_TIME : Date_And_Time;   // Date and time OB1 started
   END_VAR
   VAR_TEMP   // added for the SCL form of the ladder/FBD networks
      _w1 : Bool;
      _w2 : Bool;
      _w3 : Bool;
      _s5time1 : S5Time;
   END_VAR
BEGIN

REGION Network 1: ProcessInput
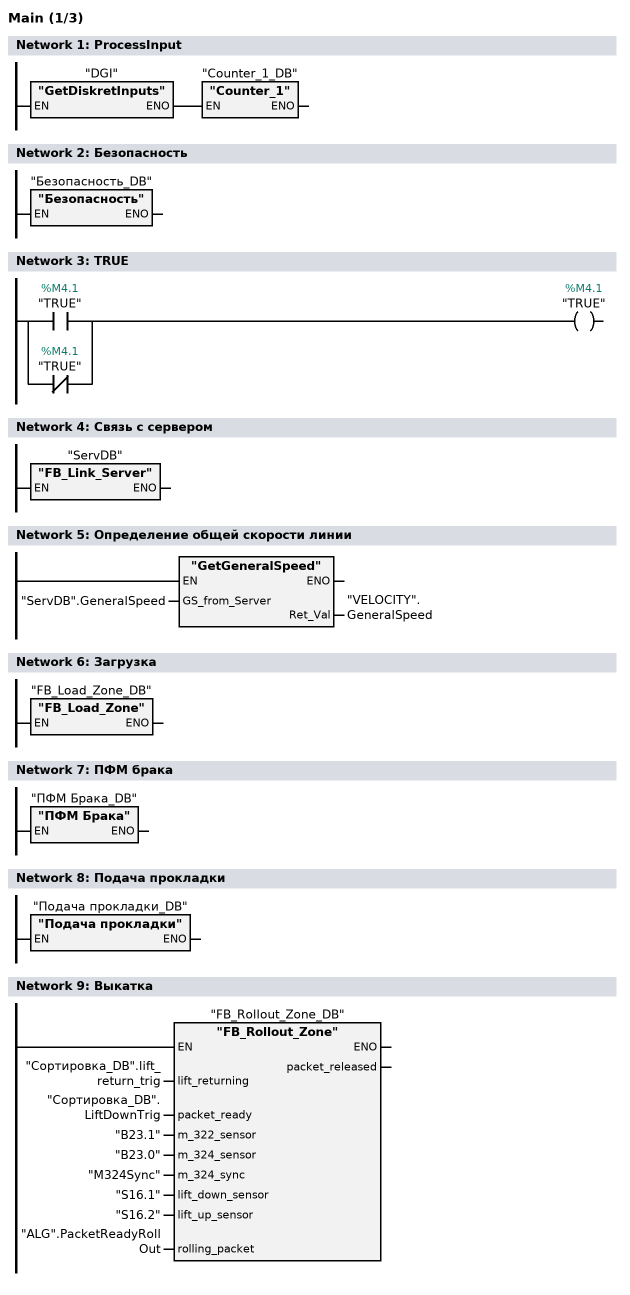
   RUNG wire#powerrail
      "DGI"()
      "Counter_1_DB"()
   END_RUNG
   // the same network as SCL:
   "DGI"(ENO => #_w1);   // "GetDiskretInputs"
   IF #_w1 THEN
       "Counter_1_DB"();   // "Counter_1"
   END_IF;
END_REGION

REGION Network 2: Безопасность
   RUNG wire#powerrail
      "Безопасность_DB"()
   END_RUNG
   // the same network as SCL:
   "Безопасность_DB"();   // "Безопасность"
END_REGION

REGION Network 3: TRUE
   RUNG wire#powerrail
      Contact( "TRUE" )
      wire#w1
      Coil( "TRUE" )
   END_RUNG
   RUNG wire#powerrail
      I_Contact( "TRUE" )
   END_RUNG wire#w1
   // the same network as SCL:
   "TRUE" := "TRUE" OR NOT "TRUE";
END_REGION

REGION Network 4: Связь с сервером
   RUNG wire#powerrail
      "ServDB"()
   END_RUNG
   // the same network as SCL:
   "ServDB"();   // "FB_Link_Server"
END_REGION

REGION Network 5: Определение общей скорости линии
   RUNG wire#powerrail
      "GetGeneralSpeed"(GS_from_Server := "ServDB".GeneralSpeed, Ret_Val => "VELOCITY".GeneralSpeed)
   END_RUNG
   // the same network as SCL:
   "VELOCITY".GeneralSpeed := "GetGeneralSpeed"(GS_from_Server := "ServDB".GeneralSpeed);
END_REGION

REGION Network 6: Загрузка
   RUNG wire#powerrail
      "FB_Load_Zone_DB"()
   END_RUNG
   // the same network as SCL:
   "FB_Load_Zone_DB"();   // "FB_Load_Zone"
END_REGION

REGION Network 7: ПФМ брака
   RUNG wire#powerrail
      "ПФМ Брака_DB"()
   END_RUNG
   // the same network as SCL:
   "ПФМ Брака_DB"();   // "ПФМ Брака"
END_REGION

REGION Network 8: Подача прокладки
   RUNG wire#powerrail
      "Подача прокладки_DB"()
   END_RUNG
   // the same network as SCL:
   "Подача прокладки_DB"();   // "Подача прокладки"
END_REGION

REGION Network 9: Выкатка
   RUNG wire#powerrail
      "FB_Rollout_Zone_DB"(lift_returning := "Сортировка_DB".lift_return_trig, packet_ready := "Сортировка_DB".LiftDownTrig, m_322_sensor := "B23.1", m_324_sensor := "B23.0", m_324_sync := "M324Sync", lift_down_sensor := "S16.1", lift_up_sensor := "S16.2", rolling_packet := "ALG".PacketReadyRollOut, packet_released =>)
   END_RUNG
   // the same network as SCL:
   "FB_Rollout_Zone_DB"(lift_returning := "Сортировка_DB".lift_return_trig,   // "FB_Rollout_Zone"
                        packet_ready := "Сортировка_DB".LiftDownTrig,
                        m_322_sensor := "B23.1",
                        m_324_sensor := "B23.0",
                        m_324_sync := "M324Sync",
                        lift_down_sensor := "S16.1",
                        lift_up_sensor := "S16.2",
                        rolling_packet := "ALG".PacketReadyRollOut);
END_REGION

REGION Network 10: Карусель прокладок
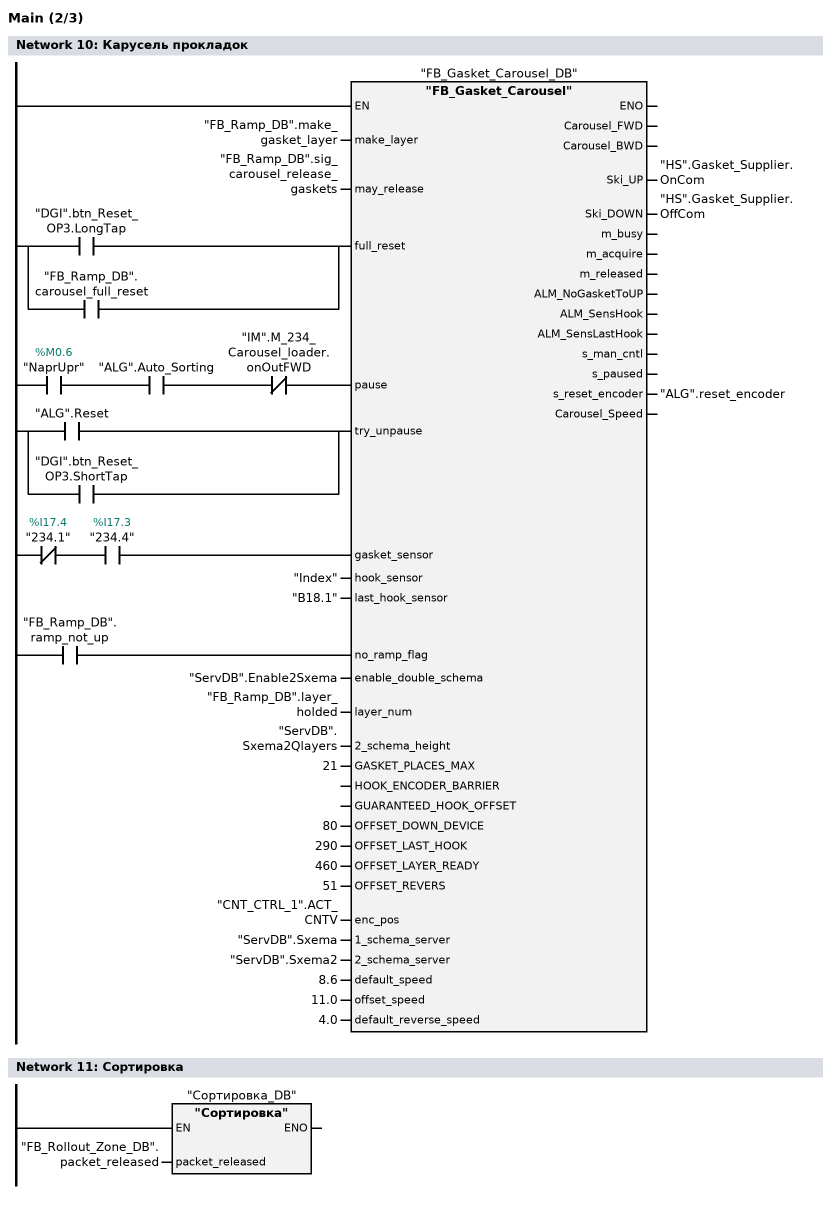
   RUNG wire#powerrail
      "FB_Gasket_Carousel_DB"(full_reset := wire#w1, pause := wire#w2, try_unpause := wire#w3, gasket_sensor := wire#w4, no_ramp_flag := wire#w5, make_layer := "FB_Ramp_DB".make_gasket_layer, may_release := "FB_Ramp_DB".sig_carousel_release_gaskets, hook_sensor := "Index", last_hook_sensor := "B18.1", enable_double_schema := "ServDB".Enable2Sxema, layer_num := "FB_Ramp_DB".layer_holded, "2_schema_height" := "ServDB".Sxema2Qlayers, GASKET_PLACES_MAX := 21, HOOK_ENCODER_BARRIER :=, GUARANTEED_HOOK_OFFSET :=, OFFSET_DOWN_DEVICE := 80, OFFSET_LAST_HOOK := 290, OFFSET_LAYER_READY := 460, OFFSET_REVERS := 51, enc_pos := "CNT_CTRL_1".ACT_CNTV, "1_schema_server" := "ServDB".Sxema, "2_schema_server" := "ServDB".Sxema2, default_speed := 8.6, offset_speed := 11.0, default_reverse_speed := 4.0, Carousel_FWD =>, Carousel_BWD =>, Ski_UP => "HS".Gasket_Supplier.OnCom, Ski_DOWN => "HS".Gasket_Supplier.OffCom, m_busy =>, m_acquire =>, m_released =>, ALM_NoGasketToUP =>, ALM_SensHook =>, ALM_SensLastHook =>, s_man_cntl =>, s_paused =>, s_reset_encoder => "ALG".reset_encoder, Carousel_Speed =>)
   END_RUNG
   RUNG wire#powerrail
      Contact( "DGI".btn_Reset_OP3.LongTap )
   END_RUNG wire#w1
   RUNG wire#powerrail
      Contact( "FB_Ramp_DB".carousel_full_reset )
   END_RUNG wire#w1
   RUNG wire#powerrail
      Contact( "NaprUpr" )
      Contact( "ALG".Auto_Sorting )
      I_Contact( "IM".M_234_Carousel_loader.onOutFWD )
   END_RUNG wire#w2
   RUNG wire#powerrail
      Contact( "ALG".Reset )
   END_RUNG wire#w3
   RUNG wire#powerrail
      Contact( "DGI".btn_Reset_OP3.ShortTap )
   END_RUNG wire#w3
   RUNG wire#powerrail
      I_Contact( "234.1" )
      Contact( "234.4" )
   END_RUNG wire#w4
   RUNG wire#powerrail
      Contact( "FB_Ramp_DB".ramp_not_up )
   END_RUNG wire#w5
   // the same network as SCL:
   "FB_Gasket_Carousel_DB"(make_layer := "FB_Ramp_DB".make_gasket_layer,   // "FB_Gasket_Carousel"
                           may_release := "FB_Ramp_DB".sig_carousel_release_gaskets,
                           full_reset := "DGI".btn_Reset_OP3.LongTap OR "FB_Ramp_DB".carousel_full_reset,
                           pause := "NaprUpr" AND "ALG".Auto_Sorting AND NOT "IM".M_234_Carousel_loader.onOutFWD,
                           try_unpause := "ALG".Reset OR "DGI".btn_Reset_OP3.ShortTap,
                           gasket_sensor := NOT "234.1" AND "234.4",
                           hook_sensor := "Index",
                           last_hook_sensor := "B18.1",
                           no_ramp_flag := "FB_Ramp_DB".ramp_not_up,
                           enable_double_schema := "ServDB".Enable2Sxema,
                           layer_num := "FB_Ramp_DB".layer_holded,
                           "2_schema_height" := "ServDB".Sxema2Qlayers,
                           GASKET_PLACES_MAX := 21,
                           OFFSET_DOWN_DEVICE := 80,
                           OFFSET_LAST_HOOK := 290,
                           OFFSET_LAYER_READY := 460,
                           OFFSET_REVERS := 51,
                           enc_pos := "CNT_CTRL_1".ACT_CNTV,
                           "1_schema_server" := "ServDB".Sxema,
                           "2_schema_server" := "ServDB".Sxema2,
                           default_speed := 8.6,
                           offset_speed := 11.0,
                           default_reverse_speed := 4.0,
                           Ski_UP => "HS".Gasket_Supplier.OnCom,
                           Ski_DOWN => "HS".Gasket_Supplier.OffCom,
                           s_reset_encoder => "ALG".reset_encoder);
END_REGION

REGION Network 11: Сортировка
   RUNG wire#powerrail
      "Сортировка_DB"(packet_released := "FB_Rollout_Zone_DB".packet_released)
   END_RUNG
   // the same network as SCL:
   "Сортировка_DB"(packet_released := "FB_Rollout_Zone_DB".packet_released);   // "Сортировка"
END_REGION

REGION Network 12: Авто режим подвижного борта
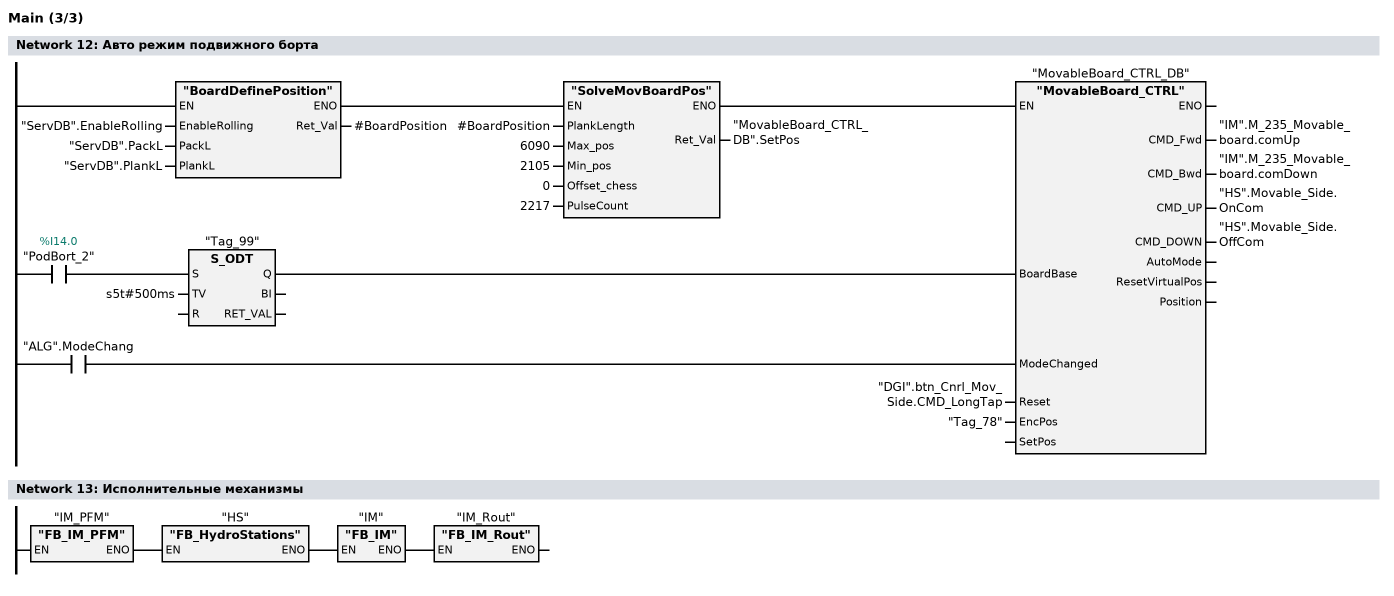
   RUNG wire#powerrail
      "BoardDefinePosition"(EnableRolling := "ServDB".EnableRolling, PackL := "ServDB".PackL, PlankL := "ServDB".PlankL, Ret_Val => #BoardPosition)
      "SolveMovBoardPos"(PlankLength := #BoardPosition, Max_pos := 6090, Min_pos := 2105, Offset_chess := 0, PulseCount := 2217, Ret_Val => "MovableBoard_CTRL_DB".SetPos)
      "MovableBoard_CTRL_DB"(BoardBase := wire#w1, ModeChanged := wire#w2, Reset := "DGI".btn_Cnrl_Mov_Side.CMD_LongTap, EncPos := "Tag_78", SetPos :=, CMD_Fwd => "IM".M_235_Movable_board.comUp, CMD_Bwd => "IM".M_235_Movable_board.comDown, CMD_UP => "HS".Movable_Side.OnCom, CMD_DOWN => "HS".Movable_Side.OffCom, AutoMode =>, ResetVirtualPos =>, Position =>)
   END_RUNG
   RUNG wire#powerrail
      Contact( "PodBort_2" )
      S_ODT(T_NO := "Tag_99", TV := s5t#500ms, R :=, BI =>, RET_VAL =>)
   END_RUNG wire#w1
   RUNG wire#powerrail
      Contact( "ALG".ModeChang )
   END_RUNG wire#w2
   // the same network as SCL:
   #BoardPosition := "BoardDefinePosition"(EnableRolling := "ServDB".EnableRolling,
                           PackL := "ServDB".PackL,
                           PlankL := "ServDB".PlankL,
                           ENO => #_w1);
   "MovableBoard_CTRL_DB".SetPos := "SolveMovBoardPos"(EN := #_w1,
                           PlankLength := #BoardPosition,
                           Max_pos := 6090,
                           Min_pos := 2105,
                           Offset_chess := 0,
                           PulseCount := 2217,
                           ENO => #_w2);
   #_s5time1 := S_ODT(T_NO := "Tag_99", S := "PodBort_2", TV := s5t#500ms, Q => #_w3);
   IF #_w2 THEN
       "MovableBoard_CTRL_DB"(BoardBase := #_w3,   // "MovableBoard_CTRL"
                              ModeChanged := "ALG".ModeChang,
                              Reset := "DGI".btn_Cnrl_Mov_Side.CMD_LongTap,
                              EncPos := "Tag_78",
                              CMD_Fwd => "IM".M_235_Movable_board.comUp,
                              CMD_Bwd => "IM".M_235_Movable_board.comDown,
                              CMD_UP => "HS".Movable_Side.OnCom,
                              CMD_DOWN => "HS".Movable_Side.OffCom);
   END_IF;
END_REGION

REGION Network 13: Исполнительные механизмы
   RUNG wire#powerrail
      "IM_PFM"()
      "HS"()
      "IM"()
      "IM_Rout"()
   END_RUNG
   // the same network as SCL:
   "IM_PFM"(ENO => #_w1);   // "FB_IM_PFM"
   "HS"(EN := #_w1, ENO => #_w2);   // "FB_HydroStations"
   "IM"(EN := #_w2, ENO => #_w3);   // "FB_IM"
   IF #_w3 THEN
       "IM_Rout"();   // "FB_IM_Rout"
   END_IF;
END_REGION
END_ORGANIZATION_BLOCK

FUNCTION_BLOCK "GetDiskretInputs"
{ S7_Optimized_Access := 'FALSE' }
VERSION : 0.1
   VAR 
      K1_1122L1 : Bool;   //    Реле безопастности К10 ОСНОВНАЯ напряжение управления
      K1_113_13L1 : Bool;   //    Реле безопастности К11 концевики группа 211,212,213,214
      K1_113_24L1 : Bool;   //    Реле безопастности К21 группа 221,222,224,225,231-235,311,312,313-317
      K1_113_35L1 : Bool;   //    Релле безопасности К31 группа 321,322,324
      k1_113_46L1 : Bool;   //    Релле безопасности К41 группа 331,332-337
      Varalla : Bool;   //    резерв
      Varalla1 : Bool;   //    резерв
      Varalla2 : Bool;   //    резерв
      F211K1_211K2 : Bool;   //    М211 включен сигналы
      F212K1 : Bool;   //    Контактор К1 Включен М212 сигналы
      F213K1 : Bool;   //    контактор К1 Включен М213 сигналы
      F214K1 : Bool;   //    М214 включен сигналы
      Varalla3 : Bool;   //    резерв
      Varalla4 : Bool;   //    резерв
      Varalla5 : Bool;   //    резерв
      Varalla6 : Bool;   //    резерв
      F221K1 : Bool;   //    М221 включен сигналы
      F222K1 : Bool;   //    Контактор К1 Включен М222 сигналы
      F223K1 : Bool;   //    Резерв
      F224K1 : Bool;   //    М224 включен сигналы
      F225K1 : Bool;   //    Контактор К1 Включен М225 сигналы
      F330K1 : Bool;   //    резерв
      Varalla8 : Bool;   //    резерв
      Varalla9 : Bool;   //    резерв
      F231K1 : Bool;   //    Контактор К1 Включен М231 сигналы
      F232K1 : Bool;   //    Контактор К1- Включен М232 сигналы
      F233K1 : Bool;   //    Контактор К1- Включен М233 сигналы
      F234K1 : Bool;   //    М234 включен сигналы
      F235K1_235K2 : Bool;   //    М235 включен сигналы
      Varalla10 : Bool;   //    резерв
      Varalla11 : Bool;   //    резерв
      Varalla12 : Bool;   //    резерв
      F311K1_311K2 : Bool;   //    М311 включен сигналы
      F312K1 : Bool;   //    М312 включен сигналы
      F313K1_313K2 : Bool;   //    М313 включен сигналы
      F314K1 : Bool;   //    М314 включен сигналы
      F315K1 : Bool;   //    М315 включен сигналы
      F316K1 : Bool;   //    М316 включен сигналы
      F317K1 : Bool;   //    Контактор К1 включен М317 сигналы
      Varalla13 : Bool;   //    резерв
      F321K1_321K2 : Bool;   //    М321 включен сигналы
      F322K1_322K2 : Bool;   //    М322 включен сигналы
      F323K1_323K2 : Bool;   //    Резерв
      F325K1 : Bool;   //    ПЧТ 324 в работе сигналы
      Varalla14 : Bool;   //    резерв
      Varalla15 : Bool;   //    резерв
      Varalla16 : Bool;   //    резеов
      Varalla17 : Bool;   //    резерв
      F331K1 : Bool;   //    М331 включен сигналы
      F332K1 : Bool;   //    Контактор К1- включен М332 сигналы
      F333K1 : Bool;   //    Контактор К1 -включен М333 сигналы
      F334K1 : Bool;   //    Контактор К1- включен М334 сигналы
      F335K1 : Bool;   //    Контактор К1- включен М335 сигналы
      F336K1 : Bool;   //    Контактор К1- включен М336 сигналы
      F337K1 : Bool;   //    резерв
      K1_323U1 : Bool;   // ПЧТ 323 в работе сигналы
      K1_221U1 : Bool;   //    ПЧТ 212 в работе сигналы
      K1_213U1 : Bool;   //    ПЧТ 213 в работе сигналы
      K1_215U1 : Bool;   //    ПЧТ 215 в работе сигналы
      K1_222U1 : Bool;   //    ПЧТ 222 в работе сигналы
      K1_225U1 : Bool;   //    Пчт 225 в работе сигналы
      K1_231U1 : Bool;   //    ПЧТ 231 в работе сигналы
      K1_233U1 : Bool;   //    ПЧТ 233 в работе сигналы
      K1_317U1 : Bool;   //    ПЧТ 317 в работе сигналы
      K1_332U1 : Bool;   //    ПЧТ 332 в работе сигналы
      K1_333U1 : Bool;   //    ПЧТ 333 в работе сигналы
      K1_334U1 : Bool;   //    ПЧТ 334 в работе сигналы
      K1_335U1 : Bool;   //    ПЧТ 335 в работе сигналы
      K1_336U1 : Bool;   //    ПЧТ 336 в работе сигналы
      K1_223U1 : Bool;   //    резерв
      K1_324U1 : Bool;   //    резерв
      K1_325U1 : Bool;   //    резерв
      K1_112_S1 : Bool;   //    Состояние концевика 112S1 сигналы
      K1_112_S2 : Bool;   //    Состояние концевика 112S2 сигналы
      K1_112_S3 : Bool;   //    Состояние концевика 112S3 сигналы
      Varalla22 : Bool;   //    резерв
      K1_113_S11 : Bool;   //    Состояние концевиков 113S11 сигналы
      K1_113_S12 : Bool;   //    Состояние концевиков 113S12 сигналы
      k1_113_S13 : Bool;   //    Состояние концевиков 113S13 сигналы
      Varalla23 : Bool;   //    резерв
      Varalla24 : Bool;   //    резерв
      FC_223_1 : Bool;   // начало зоны оценки
      FC_223_2 : Bool;   //  конец зоны оценки
      FC_223_3 : Bool;   // сброс после зоны оценки
      Varalla28 : Bool;   //    резерв
      Varalla29 : Bool;   //    резерв
      Varalla30 : Bool;   //    резерв
      Varalla31 : Bool;   //    резерв
      Liftdown : Bool;   //    Лифт вниз
      LiftUp : Bool;   //    Лифт в верх
      sloidoski : Bool;   //    Слой доски 1
      sloidoski2 : Bool;   //    Слой доски 2
      doskavpriymkeelevator : Bool;   //    Доска в приямке элеватора
      koncevik1 : Bool;   //    концевик 1(середина приемного транспортера)
      koncevik2 : Bool;   //    концевик 2 (вилы лифта приемного транспортера)
      nakloniytransporter : Bool;   //    наклонный транспортер датчик
      FC_18_Length : Bool;   //    FC18. Сортировка. Линейка длины. 1.8 м
      F2_1m : Bool;   //    F2,1 длинна
      F2_4m : Bool;   //    F2,4 длинна
      F2_7m : Bool;   //    F2,7 длинна
      F3_0m : Bool;   //    F3,0 длинна
      F3_3m : Bool;   //    F3,3 длинна
      F3_6m : Bool;   //    F3,6 длинна
      F3_9m : Bool;   //    F3,9 длинна
      F4_2m : Bool;   //    F4,2 длинна
      F4_5m : Bool;   //    F4,5 длинна
      F4_8m : Bool;   //    F4,8 длинна
      F5_1m : Bool;   //    F5,1 длинна
      F5_4m : Bool;   //    F5,4 длинна
      F5_7m : Bool;   //    F5,7 длинна
      F6_0m : Bool;   //    F6,0 длинна
      PodBort_1 : Bool;   //    резерв
      PodBort_2 : Bool;
      "312Alarm" : Bool;   // ошибка ПЧТ 312
      S14_2 : Bool;   //    Максимальная ширина доски концевик М225 зона
      S14_3 : Bool;   //    Минимальная ширина доски концевик М225 зона
      B14_4 : Bool;   //    счет доски М225 зона после бобышек
      B14_5 : Bool;   //    счет доски М225 зона после бобышек
      K1_312U1 : Bool;   // ПЧТ 312 в работе сигналы
      S14_7 : Bool;   //    заднее положение вил
      S15_0 : Bool;   //    замедление вил назад
      S15_1 : Bool;   //    замедление в перед вил
      S15_2 : Bool;   //    Переднее положение вил
      reserv5 : Bool;   //    резерв
      Index : Bool;   //    резерв
      B15_5 : Bool;   //    вилы в низу
      B15_6 : Bool;   //    вилы ожидание
      B15_7 : Bool;   //    вилы в верху
      FC_232_1 : Bool;   //    набор слоя пакета на лифте
      S16_1 : Bool;   //    лифт ПфМ в низу
      S16_2 : Bool;   //    лифт ПФМ в верху
      E16_3 : Bool;   //    Температура гидростанции
      E16_4 : Bool;   //    Уровень Гидростанции
      FC_232_2 : Bool;   // набор слоя пакета на лифте
      B16_6 : Bool;   //    верхнее положение упоров на рольганге
      S16_7 : Bool;   //    нижнее положение упоров на рольганге
      B17_0 : Bool;   //    наличие прокладок на М313
      B17_1 : Bool;   //    наличие прокладки в М314
      B17_2 : Bool;   //    наличие прокладки в М315
      B17_3 : Bool;   //    резерв
      B17_4 : Bool;   //    резерв
      Varalla32 : Bool;   //    резерв
      Varalla33 : Bool;   //    резерв
      Varalla34 : Bool;   //    резерв
      B18_0 : Bool;   //    рейкоукладчик в низу
      B18_1 : Bool;   //    рейкоукладчик в верху
      S18_2 : Bool;   //    позиция рамы 1
      S18_3 : Bool;   //    позиция рамы 2
      B18_4 : Bool;   //    датчик положения захвата прокладки открыто
      B18_5 : Bool;   //    датчик положени захвата прокладки закрыто
      B18_6 : Bool;   //    замедление транспортера прокладок
      B18_7 : Bool;   //    Остановка транспортера прокладок
      B19_0 : Bool;   //    Обратный ход транспортера прокладок ДАТЧИК
      Varalla35 : Bool;   //    резерв
      Varalla36 : Bool;   //    резерв
      Varalla37 : Bool;   //    резерв
      Varalla38 : Bool;   //    резерв
      Varalla39 : Bool;   //    резерв
      Varalla40 : Bool;   //    резерв
      Varalla41 : Bool;   //    резерв
      Varalla42 : Bool;   //    резерв
      Varalla43 : Bool;   //    резерв
      Varalla44 : Bool;   //    резерв
      Varalla45 : Bool;   //    резерв
      Varalla46 : Bool;   //    резерв
      Varalla47 : Bool;   //    резерв
      Varalla48 : Bool;   //    резерв
      Varalla49 : Bool;   //    резерв
      Varalla50 : Bool;   //    резерв
      Varalla51 : Bool;   //    резерв
      Varalla52 : Bool;   //    резерв
      Varalla53 : Bool;   //    резерв
      Varalla54 : Bool;   //    резерв
      Varalla55 : Bool;   //    резерв
      Varalla56 : Bool;   //    резерв
      Varalla57 : Bool;   //    резерв
      B22_0 : Bool;   //    доска в конце роликового транспортера(брак)
      B22_1 : Bool;   //    доска в начале роликового транспортера(брак)
      S22_2 : Bool;   //    вилы брака ПФМ в перед
      S22_3 : Bool;   //    вилы брака ПФМ назад
      B22_4 : Bool;   //    лифт брака ПФМ в верху
      B22_5 : Bool;   //    лифт брака ПФМ в низу
      B22_6 : Bool;   //    Слой на вилах брака ПФМ
      FC_22_7 : Bool;   // Счет досок в слое
      B23_0 : Bool;   //    непонятно
      B23_1 : Bool;   //    пакет на разгрузочном транспортере 3024
      Varalla59 : Bool;   //    резерв
      Varalla60 : Bool;   //    резерв
      Varalla61 : Bool;   //    резерв
      Varalla62 : Bool;   //    резерв
      FC_23_6 : Bool;   //    резерв
      FC_23_7 : Bool;   //    резерв
      S76 : Bool;   //    стоповая кнопка OP1
      S76_1 : Bool;   //    Включение напряжения управления
      S76_2 : Bool;   //    Подтверждение ошибки
      S76_3 : Bool;   //    Гидравлика линии в положении включено
      E76_4 : Bool;   //    Старт гидравлики
      S76_5 : Bool;   //    авто включение и выключение загрузчика ( режим авто всей загрузки)
      S76_6 : Bool;   //    авто М211 приемный транспортер
      E76_7 : Bool;   //    вперед М211 приемный транспортер в автомате
      S77_0 : Bool;   //    авто М221 горка
      E77_1 : Bool;   //    вперед М221 горка в автомате
      S77_2 : Bool;   //    Квитирование зоны 1(от горки до ПФМ)
      S77_3 : Bool;   //    Квитирование зоны выгрузки
      S77_4 : Bool;   //    Квитирование зоны 2  (ПФМ брака)
      S77_5 : Bool;   //    авто режим зоны 1( включено, выключено) ( от горки до ПФМ)
      S77_6 : Bool;   //    Выдвинуть упоры поштучника
      E77_7 : Bool;   //    Убрать упоры поштучника
      S78_0 : Bool;   //    Вилы выдвинуть
      E78_1 : Bool;   //    Вилы задвинуть
      S78_2 : Bool;   //    Вилы опустить
      E78_3 : Bool;   //    Вилы поднять
      S78_4 : Bool;   //    Лифт опустить
      E78_5 : Bool;   //    Лифт поднять
      S78_6 : Bool;   //    рейкоукладчик вниз
      E78_7 : Bool;   //    рейкоукладчик вверх
      S79_0 : Bool;   //    0
      S79_1 : Bool;   //    авто подача прокладки(включен,выключен)
      E79_2 : Bool;   //    резерв
      S79_3 : Bool;   //    авто режим ПФМ брака (включено,выключено)
      S79_4 : Bool;   //    Сброс с рольганга(брака) вперпед
      S79_5 : Bool;   //    Транспортер набора слоя ( брака) вперед
      S79_6 : Bool;   //    вилы( брака) вперед
      E79_7 : Bool;   //    вилы( брака) назад
      S80_0 : Bool;   //    опустить вилы ПФМ( брака)
      E80_1 : Bool;   //    поднять вилы ПФМ( брака)
      S80_2 : Bool;   //    Лифт ПФМ(брака) опустить
      E80_3 : Bool;   //    Лифт ПФМ(брака) поднять
      S80_4 : Bool;   //    поднять, опустить Подвижный борт(М235)
      S80_5 : Bool;   //    вперед подвижный борт(М235)
      E80_6 : Bool;   //    назад подвижный борт(М235)
      S80_7 : Bool;   //    0
      Varalla106 : Bool;   //    резерв
      Varalla107 : Bool;   //    резерв
      Varalla108 : Bool;   //    резерв
      Varalla109 : Bool;   //    резерв
      Varalla110 : Bool;   //    резерв
      Varalla111 : Bool;   //    резерв
      Varalla112 : Bool;   //    резерв
      Varalla113 : Bool;   //    резерв
      S82_0 : Bool;   //    Стоп ОР2
      S81_1 : Bool;   //    Приемный транспортер вперед ОР2
      E82_2 : Bool;   //    Приемный транспортер назад ОР2
      S82_3 : Bool;   //    Авто загрузка включена,выключена ОР2
      S82_4 : Bool;   //    Лифт загрузки поднять ОР2
      E82_5 : Bool;   //    Лифт загрузки опустить ОР2
      S82_6 : Bool;   //    Наклонный транспортер авто ОР2
      E82_7 : Bool;   //    Авто наклонный транспортер вперед ОР2
      S83_0 : Bool;   //    Ленточный транспортер удаления прокладок назад ОР2
      E83_1 : Bool;   //    Ленточный транспортер удаления прокладок вперед ОР2
      E83_2 : Bool;   //    Горка прокладок 1 авто ОР2
      E83_3 : Bool;   //    Горка прокладок 1 вперед ОР2(авто)
      S83_4 : Bool;   //    Квитирование зоны 1 ОР2
      Varalla114 : Bool;   //    резерв
      Varalla115 : Bool;   //    резерв
      Varalla116 : Bool;   //    резерв
      S84_0 : Bool;   //    Стоп ОР3
      S84_1 : Bool;   //    Транспортер М317 прокладок вперед ОР3
      E84_2 : Bool;   //    Транспортер М317 прокладок назад ОР3
      S84_3 : Bool;   //    Дозировани включено ОР3
      S84_4 : Bool;   //    авто подача прокладок включена, выключена ОР3
      S84_5 : Bool;   //    Рейкоукладчик вниз ОР3
      E84_6 : Bool;   //    Рейкоукладчик вверх ОР3
      S84_7 : Bool;   //    Открыть стакан прокладки ОР3
      E85_0 : Bool;   //    Закрыть стакан прокладки ОР3
      S85_1 : Bool;   //    0
      E85_2 : Bool;   //    0
      S85_3 : Bool;   //    авто горка прокладок 2,3 ОР3
      E85_4 : Bool;   //    горка 2,3 прокладок вперед(авто) ОР3
      S85_5 : Bool;   //    М234 назад ОР3
      E85_6 : Bool;   //    М234 вперед транспортер прокладок перед крючками ОР3
      S85_7 : Bool;   //    Квитирование зоны прокладок ОР3
      S86_0 : Bool;   //    Лифт ПФМ вниз ОР3
      E86_1 : Bool;   //    ЛИфт ПФМ вверх ОР3
      S86_2 : Bool;   //    Ролики лифта ПФМ вперед ОР3
      S86_3 : Bool;   //    ПФМ Основное Авто включено, выключено ОР3
      S86_4 : Bool;   //    Подтверждение неисправности ОР3
      S86_5 : Bool;   //    датчик
      Varalla117 : Bool;   //    резерв
      Varalla118 : Bool;   //    резерв
      S87_0 : Bool;   //    Кнопка брака ОР1.1
      S87_1 : Bool;   //    Горка авто ОР1.1
      E87_2 : Bool;   //    Горка ОР1.1 (авто)
      S87_3 : Bool;   //    педаль 1ОР1.1
      S87_4 : Bool;   //    педаль2 ОР1.1
      Varalla119 : Bool;   //    резерв
      Varalla120 : Bool;   //    резерв
      Varalla121 : Bool;   //    резерв
      S88_0 : Bool;   //    Стоп ОР4
      K3_3 : Bool;   //    работа подвижного борта ОР4
      S88_2 : Bool;   //    Выкатной транспортер 1 ПФМ назад ОР4
      E88_3 : Bool;   //    Выкатной транспортер 1 ПФМ вперед ОР4
      S88_4 : Bool;   //    Выкатной транспортер 2 ПФМ назад ОР4
      S88_5 : Bool;   //    Выкатной транспортер 2 ПФМ вперед ОР4
      E88_6 : Bool;   //    резерв ОР4
      S88_7 : Bool;   //    резерв ОР4
      S89_0 : Bool;   //    Выкатной транспортер 4 ПФМ назад ОР4
      S89_1 : Bool;   //    Выкатной транспортер 4 ПФМ вперед ОР4
      S89_2 : Bool;   //    Квитирование ОР4
      S89_3 : Bool;   //    датчик ОР4
      Varalla122 : Bool;   //    резерв ОР4
      Varalla123 : Bool;   //    резерв ОР4
      Varalla124 : Bool;   //    резерв ОР4
      Varalla125 : Bool;   //    резерв ОР4
      S90_0 : Bool;   //    Стоп ОР5
      S90_1 : Bool;   //    М331 вперед ленточный транспортер брака ОР5
      S90_2 : Bool;   //    М332 вперед сбрасыватель рольганга брака ОР5
      Varalla126 : Bool;   //    резерв
      S90_4 : Bool;   //    Вилы ПФМ брака назад ОР5
      E90_5 : Bool;   //    Вилы ПФМ брака вперед ОР5
      S90_6 : Bool;   //    Опустить упоры формирования слоя на ПФМ брака ОР5
      E90_7 : Bool;   //    Поднять упоры формирования слоя на ПФМ брака ОР5
      S91_0 : Bool;   //    Лифт брака ПФМ опустить ОР5
      E91_1 : Bool;   //    Лифт брака ПФМ поднять ОР5
      S91_2 : Bool;   //    квитирование ПФМ 2
      Varalla127 : Bool;   //    резерв
      Varalla128 : Bool;   //    резерв
      Varalla129 : Bool;   //    резерв
      Varalla130 : Bool;   //    резерв
      Varalla131 : Bool;   //    резерв
      S214 : Bool;   // пуск стоп приемного транспортера прокладок
      BrakDroper_front : Bool;
      BrakDroppperBob_old : Bool;
      UporDefectivePFM_timer {InstructionName := 'TON'; LibVersion := '1.0'; S7_SetPoint := 'False'} : TON;   // дожимщик для упоров пфм брака
      GasketRampSqueeze_timer {InstructionName := 'TON'; LibVersion := '1.0'} : TON;   // дожимщик для рамы прокладок
      TopSig_timer {InstructionName := 'TON'; LibVersion := '1.0'} : TON;   // дожимщик верхнего положения рамы прокладок
      PFMdefect_vill_fwd {InstructionName := 'TON'; LibVersion := '1.0'} : TON;
      MidSig_timer {InstructionName := 'TOF'; LibVersion := '1.0'} : TOF;   // дожимщик для среднего положения
      SensHook_timer {InstructionName := 'TOF'; LibVersion := '1.0'} : TOF;
      SensHookDovod_timer {InstructionName := 'TOF'; LibVersion := '1.0'} : TOF;
      SensStartEvalZone_timer {InstructionName := 'TOF'; LibVersion := '1.0'} : TOF;   // начало зоны оценки
      SensEndEvalZone_timer {InstructionName := 'TON'; LibVersion := '1.0'} : TON;   // конец зоны оценки
      SensDropDefect_timer {InstructionName := 'TOF'; LibVersion := '1.0'} : TOF;   // сброс в брак 
      SensBoardCounter_timer {InstructionName := 'TOF'; LibVersion := '1.0'} : TOF;   // счет досок в слое ПФМ брака
      SensBoardCounterFilter_timer {InstructionName := 'TON'; LibVersion := '1.0'} : TON;   // фильтр на счет ПФМ брака
      SensNewBobBrak_timer {InstructionName := 'TOF'; LibVersion := '1.0'} : TOF;   // датчик новой бобышки на пфм брака
      btn_Drop_Defect { S7_SetPoint := 'False'} : "Button_ShortTap";   // кнопка контроля сброса брака
      "btn_Stop_M331/330" : "Button_ShortTap";   // кнопка выключения транспортера сброса в брак
      btn_btnLenta_defect : "Button_ShortTap";   // кнопка включения/выключения ленты брака 
      btn_Force_Finish : "Button_ShortTap";   // кнопка принудительного завершения сборки пакета
      btn_DropFromRollerDefect : "Button_ShortTap";   // кнопка сброса с рольганга брака
      btn_Cnrl_Mov_Side { S7_SetPoint := 'False'} : "ButtonSwitcher_PlusLongTap";   // кнопка контроля подвижного борта (вверх/вниз)
      btn_Auto_Loading : "ButtonSwitcher";   // кнопка переключения авторежима загрузки
      btn_Auto_Sorting : "ButtonSwitcher";   // кнопка переключения авторежима сортировки
      btn_Auto_Gasket : "ButtonSwitcher";   // кнопка переключения авторежима на подаче прокладки
      btn_Auto_PFM_defective : "ButtonSwitcher";   // кнопка переключения авторежима ПФМ брака
      btn_Reset_OP3 : "ButtonShortLongTap";   // кнопка сброса ошибки на пульте OP3
      btn_ResetUporLine : "Button_PlusLongTap";   // кнопка обновления задания упоров и сброса калибровки линейки
   END_VAR


BEGIN
	
	#K1_1122L1 := "K1-112 2L1"; //Реле безопастности К10 ОСНОВНАЯ напряжение управления
	#K1_113_13L1 := "K1-113/1 3L1"; //Реле безопастности К11 концевики группа 211,212,213,214
	#K1_113_24L1 := "K1-113/2 4L1"; //Реле безопастности К21 группа 221,222,224,225,231-235,311,312,313-317
	#K1_113_35L1 := "K1-113/3 5L1"; //Релле безопасности К31 группа 321,322,324
	#k1_113_46L1 := "k1-113/4 6L1"; //Релле безопасности К41 группа 331,332-337
	#Varalla := "Varalla"; //резерв
	#Varalla1 := "Varalla1"; //резерв
	#Varalla2 := "Varalla2"; //резерв
	#F211K1_211K2 := "211K1/211K2"; //М211 включен сигналы
	#F212K1 := "212K1"; //Контактор К1 Включен М212 сигналы
	#F213K1 := "213K1"; //контактор К1 Включен М213 сигналы
	#F214K1 := "214K1"; //М214 включен сигналы
	#Varalla3 := "Varalla3"; //резерв
	#Varalla4 := "Varalla4"; //резерв
	#Varalla5 := "Varalla5"; //резерв
	#Varalla6 := "Varalla6"; //резерв
	#F221K1 := "221K1"; //М221 включен сигналы
	#F222K1 := "222K1"; //Контактор К1 Включен М222 сигналы
	#F223K1 := "223K1"; //Резерв
	#F224K1 := "224K1"; //М224 включен сигналы
	#F225K1 := "225K1"; //Контактор К1 Включен М225 сигналы
	#F330K1 := "330K1"; //резерв
	#Varalla8 := "Varalla8"; //резерв
	#Varalla9 := "Varalla9"; //резерв
	#F231K1 := "231K1"; //Контактор К1 Включен М231 сигналы
	#F232K1 := "232K1"; //Контактор К1- Включен М232 сигналы
	#F233K1 := "233K1"; //Контактор К1- Включен М233 сигналы
	#F234K1 := "234K1"; //М234 включен сигналы
	#F235K1_235K2 := "235K1/235K2"; //М235 включен сигналы
	#Varalla10 := "Varalla10"; //резерв
	#Varalla11 := "Varalla11"; //резерв
	#Varalla12 := "Varalla12"; //резерв
	#F311K1_311K2 := "311K1/311K2"; //М311 включен сигналы
	#F312K1 := "312K1"; //М312 включен сигналы
	#F313K1_313K2 := "313K1/313K2"; //М313 включен сигналы
	#F314K1 := "314K1"; //М314 включен сигналы
	#F315K1 := "315K1"; //М315 включен сигналы
	#F316K1 := "316K1"; //М316 включен сигналы
	#F317K1 := "317K1"; //Контактор К1 включен М317 сигналы
	#Varalla13 := "Varalla13"; //резерв
	#F321K1_321K2 := "321K1/321K2"; //М321 включен сигналы
	#F322K1_322K2 := "322K1/322K2"; //М322 включен сигналы
	#F323K1_323K2 := "323K1/323K2"; //Резерв
	#F325K1 := "325K1"; //ПЧТ 325 в работе сигналы
	#Varalla14 := "K1-324U.1"; //резерв
	#Varalla15 := "Varalla15"; //резерв
	#Varalla16 := "Varalla16"; //резеов
	#Varalla17 := "Varalla17"; //резерв
	#F331K1 := "331K1"; //М331 включен сигналы
	#F332K1 := "332K1"; //Контактор К1- включен М332 сигналы
	#F333K1 := "333K1"; //Контактор К1 -включен М333 сигналы
	#F334K1 := "334K1"; //Контактор К1- включен М334 сигналы
	#F335K1 := "335K1"; //Контактор К1- включен М335 сигналы
	#F336K1 := "336K1"; //Контактор К1- включен М336 сигналы
	#F337K1 := "337K1"; //резерв
	#K1_323U1 := "K1-323U1"; //резерв
	#K1_221U1 := "K1-212U1"; //ПЧТ 212 в работе сигналы
	#K1_213U1 := "K1-213U1"; //ПЧТ 213 в работе сигналы
	#K1_215U1 := "K1-215U1"; //ПЧТ 215 в работе сигналы
	#K1_222U1 := "K1-222U1"; //ПЧТ 222 в работе сигналы
	#K1_225U1 := "K1-225U1"; //Пчт 225 в работе сигналы
	#K1_231U1 := "K1-231U1"; //ПЧТ 231 в работе сигналы
	#K1_233U1 := "K1-233U1"; //ПЧТ 233 в работе сигналы
	#K1_317U1 := "K1-317U1"; //ПЧТ 317 в работе сигналы
	#K1_332U1 := "K1-332U1"; //ПЧТ 332 в работе сигналы
	#K1_333U1 := "K1-333U1"; //ПЧТ 333 в работе сигналы
	#K1_334U1 := "K1-334U1"; //ПЧТ 334 в работе сигналы
	#K1_335U1 := "K1-335U1"; //ПЧТ 335 в работе сигналы
	#K1_336U1 := "K1-336U1"; //ПЧТ 336 в работе сигналы
	#K1_223U1 := "K1-223U1"; //ПЧТ 223 в работе сигналы
	#K1_324U1 := "K1-324U1"; //ПЧТ 324 в работе сигналы
	#K1_325U1 := "K1-325U1"; //ПЧТ 325 в работе сигналы
	#K1_112_S1 := "K1/112-S1"; //Состояние концевика 112S1 сигналы
	#K1_112_S2 := "K1/112-S2"; //Состояние концевика 112S2 сигналы
	#K1_112_S3 := "K1/112-S3"; //Состояние концевика 112S3 сигналы
	#Varalla22 := "Varalla22"; //резерв
	#K1_113_S11 := "K1/113-S11"; //Состояние концевиков 113S11 сигналы
	#K1_113_S12 := "K1/113-S12"; //Состояние концевиков 113S12 сигналы
	#k1_113_S13 := "k1/113-S13"; //Состояние концевиков 113S13 сигналы
	#Varalla23 := "FC 323.1"; //резерв
	#Varalla24 := "FC 323.2"; //резерв
	
	#SensStartEvalZone_timer(IN := "FC 223.1",
	                         PT := T#500ms
	);
	
	#FC_223_1 := #SensStartEvalZone_timer.Q; //начало зоны оценки
	
	#SensEndEvalZone_timer(IN:="FC 223.2",
	                       PT:=T#200ms);
	
	#FC_223_2 := #SensEndEvalZone_timer.Q; //конец зоны оценки
	
	#SensDropDefect_timer(IN:="FC 223.3",
	                      PT:=T#500ms);
	
	#FC_223_3 := #SensDropDefect_timer.Q ; //сброс в брак
	
	#Varalla28 := "FC_323_1"; //резерв
	#Varalla29 := "Key_Faser"; //резерв
	#Varalla30 := "Varalla30"; //резерв
	#Varalla31 := "Varalla31"; //резерв
	#Liftdown := "Lift Upp"; //Лифт вниз
	#LiftUp := "Lift Down"; //Лифт в верх
	#sloidoski := "sloi doski"; //Слой доски 1
	#sloidoski2 := "sloi doski2"; //Слой доски 2
	#doskavpriymkeelevator := "doska v priymke elevator"; //Доска в приямке элеватора
	#koncevik1 := "koncevik1"; //концевик 1(середина приемного транспортера)
	#koncevik2 := "koncevik2"; //концевик 2 (вилы лифта приемного транспортера)
	#nakloniytransporter := "nakloniy transporter"; //наклонный транспортер датчик
	#FC_18_Length := "1,8m"; //FC18. Сортировка. Линейка длины. 1.8 м
	#F2_1m := "2,1m"; //F2,1 длинна
	#F2_4m := "2,4m"; //F2,4 длинна
	#F2_7m := "2,7m"; //F2,7 длинна
	#F3_0m := "3,0m"; //F3,0 длинна
	#F3_3m := "3,3m"; //F3,3 длинна
	#F3_6m := "3,6m"; //F3,6 длинна
	#F3_9m := "3,9m"; //F3,9 длинна
	#F4_2m := "4,2m"; //F4,2 длинна
	#F4_5m := "4,5m"; //F4,5 длинна
	#F4_8m := "4,8m"; //F4,8 длинна
	#F5_1m := "5,1m"; //F5,1 длинна
	#F5_4m := "5,4m"; //F5,4 длинна
	#F5_7m := "5,7m"; //F5,7 длинна
	#F6_0m := "6,0m"; //F6,0 длинна
	#PodBort_1 := "PodBort_1"; //резерв
	#PodBort_2 := "PodBort_2";
	#"312Alarm" := "K312Fault"; //индуктивные датчики 2 М225( поштучник) кейфазер2
	#S14_2 := "S14.2"; //Максимальная ширина доски концевик М225 зона
	#S14_3 := "S14.3"; //Минимальная ширина доски концевик М225 зона
	#B14_4 := "B14.4"; //счет доски М225 зона после бобышек
	#B14_5 := "B14.5"; //счет доски М225 зона после бобышек
	#K1_312U1 := "K-312U1"; //счет доски М225 зона после бобышек
	#S14_7 := "S14.7"; //заднее положение вил
	#S15_0 := "S15.0"; //замедление вил назад
	#S15_1 := "S15.1"; //замедление в перед вил
	#S15_2 := "S15.2"; //Переднее положение вил
	#reserv5 := "311_S1"; //резерв
	#B15_5 := "B15.5"; //вилы в низу
	#B15_6 := "311_S2"; //вилы ожидание
	#B15_7 := "B15.7"; //вилы в верху
	#FC_232_1 := "FC_232_1"; //набор слоя пакета на лифте
	#S16_1 := "S16.1"; //лифт ПфМ в низу
	#S16_2 := "S16.2"; //лифт ПФМ в верху
	#E16_3 := "FC_225_Upor"; //Температура гидростанции
	#E16_4 := "E16.4"; //Уровень Гидростанции
	#FC_232_2 := "FC_232_2"; //набор слоя пакета на лифте
	#B16_6 := "KeyFazerPFM_repeater"; //верхнее положение упоров на рольганге
	#S16_7 := "KeyFazerPFM"; //нижнее положение упоров на рольганге
	#B17_0 := "B17.0"; //наличие прокладок на М313
	#B17_1 := "B17.1"; //наличие прокладки в М314
	#B17_2 := "B17.2"; //наличие прокладки в М315
	#B17_3 := "234.4"; //резерв
	#B17_4 := "234.1"; //резерв
	#Varalla32 := "234.2"; //резерв
	#Varalla33 := "234.3"; //резерв
	#Varalla34 := "Fc316"; //резерв
	
	#TopSig_timer(IN:="B18.0",
	              PT:=T#160ms);
	#B18_0 := #TopSig_timer.Q; //рейкоукладчик вверху
	
	#MidSig_timer(IN := "S18.2",
	              PT := T#500ms);
	#S18_2 := #MidSig_timer.Q; //позиция рамы 1
	
	#S18_3 := "S18.3"; //позиция рамы 2
	#GasketRampSqueeze_timer(IN:="S18.3",
	                         PT:="ALG".SqueezeRamp);
	
	
	#SensHook_timer(IN:="Index",
	                PT:=T#300ms);
	
	#Index := #SensHook_timer.Q;
	
	#SensHookDovod_timer(IN:="B18.1",
	                     PT:=T#300ms);
	
	#B18_1 := #SensHookDovod_timer.Q;
	
	#B18_4 := "B18.4"; //датчик положения захвата прокладки открыто
	#B18_5 := "B18.5"; //датчик положени захвата прокладки закрыто
	#B18_6 := "B18.6"; //замедление транспортера прокладок
	#B18_7 := "B18.7"; //Остановка транспортера прокладок
	#B19_0 := "B19.0"; //Обратный ход транспортера прокладок ДАТЧИК
	#Varalla35 := "Varalla35"; //резерв
	#Varalla36 := "Varalla36"; //резерв
	#Varalla37 := "Varalla37"; //резерв
	#Varalla38 := "Varalla38"; //резерв
	#Varalla39 := "Varalla39"; //резерв
	#Varalla40 := "Varalla40"; //резерв
	#Varalla41 := "Varalla41"; //резерв
	#Varalla42 := "Varalla42"; //резерв
	#Varalla43 := "Varalla43"; //резерв
	#Varalla44 := "Varalla44"; //резерв
	#Varalla45 := "Varalla45"; //резерв
	#Varalla46 := "Varalla46"; //резерв
	#Varalla47 := "Varalla47"; //резерв
	#Varalla48 := "Varalla48"; //резерв
	#Varalla49 := "Varalla49"; //резерв
	#Varalla50 := "Varalla50"; //резерв
	#Varalla51 := "Varalla51"; //резерв
	#Varalla52 := "Varalla52"; //резерв
	#Varalla53 := "Varalla53"; //резерв
	#Varalla54 := "Varalla54"; //резерв
	#Varalla55 := "Varalla55"; //резерв
	#Varalla56 := "Varalla56"; //резерв
	#Varalla57 := "Varalla57"; //резерв
	#B22_0 := "B22.0"; //доска в конце роликового транспортера(брак)
	
	
	#SensNewBobBrak_timer(IN:="B22.1",
	                      PT:=T#1s);
	#B22_1 := #SensNewBobBrak_timer.Q; //доска в начале роликового транспортера(брак)
	// выдаем фронт сигнала
	// 
	#BrakDroper_front := #B22_1 AND NOT #BrakDroppperBob_old;
	#BrakDroppperBob_old := #B22_1;
	
	#S22_2 := "S22.2"; //вилы брака ПФМ в перед
	#S22_3 := "S22.3"; //вилы брака ПФМ назад
	#B22_4 := "B22.4"; //лифт брака ПФМ в верху
	#B22_5 := "B22.5"; //лифт брака ПФМ в низу
	#B22_6 := "B22.6"; //Слой на вилах брака ПФМ
	
	
	#SensBoardCounterFilter_timer(IN:="FC 22.7",
	                              PT:=T#100ms
	);
	
	#SensBoardCounter_timer(IN := #SensBoardCounterFilter_timer.Q,
	                        PT := T#500ms);
	
	#FC_22_7 := #SensBoardCounter_timer.Q; // счет досок в слое ПФМ брака
	
	#B23_0 := "B23.0"; //непонятно
	#B23_1 := "B23.1"; //пакет на разгрузочном транспортере 3024
	#Varalla59 := "M324Sync"; //резерв
	#Varalla60 := "Varalla60"; //резерв
	#Varalla61 := "Varalla61"; //резерв
	#Varalla62 := "Varalla62"; //резерв
	
	#UporDefectivePFM_timer(IN:="FC 23.6" OR "FC 23.7",
	                        PT:=T#1500ms);
	
	#FC_23_6 := "FC 23.6" AND #UporDefectivePFM_timer.Q; //резерв
	#FC_23_7 := "FC 23.7" AND #UporDefectivePFM_timer.Q; //резерв
	#S76 := "S76"; //стоповая кнопка OP1
	#S76_1 := "S76.1"; //Включение напряжения управления
	#S76_2 := "S76.2"; //Подтверждение ошибки
	#S76_3 := "S76.3"; //Гидравлика линии в положении включено
	#E76_4 := "E76.4"; //Старт гидравлики
	#S76_5 := "S76.5"; //авто включение и выключение загрузчика ( режим авто всей загрузки)
	#S76_6 := "S76.6"; //авто М211 приемный транспортер
	#E76_7 := "E76.7"; //вперед М211 приемный транспортер в автомате
	#S77_0 := "S77.0"; //авто М221 горка
	#E77_1 := "E77.1"; //вперед М221 горка в автомате
	#S77_2 := "S77.2"; //Квитирование зоны 1(от горки до ПФМ)
	#S77_3 := "S77.3"; //Квитирование зоны выгрузки
	#S77_4 := "S77.4"; //Квитирование зоны 2  (ПФМ брака)
	#S77_5 := "S77.5"; //авто режим зоны 1( включено, выключено) ( от горки до ПФМ)
	#S77_6 := "S77.6"; //Выдвинуть упоры поштучника
	#E77_7 := "E77.7"; //Убрать упоры поштучника
	#S78_0 := "S78.0"; //Вилы выдвинуть
	#E78_1 := "E78.1"; //Вилы задвинуть
	#S78_2 := "S78.2"; //Вилы опустить
	#E78_3 := "E78.3"; //Вилы поднять
	#S78_4 := "S78.4"; //Лифт опустить
	#E78_5 := "E78.5"; //Лифт поднять
	#S78_6 := "S78.6"; //рейкоукладчик вниз
	#E78_7 := "E78.7"; //рейкоукладчик вверх
	#S79_0 := "S79.0"; //0
	#S79_1 := "S79.1"; //авто подача прокладки(включен,выключен)
	#E79_2 := "E79.2"; //резерв
	#S79_3 := "S79.3"; //авто режим ПФМ брака (включено,выключено)
	
	#btn_DropFromRollerDefect(Sig := "S79.4",
	                          set_Response_Time := T#70ms);
	#S79_4 := #btn_DropFromRollerDefect.Out; //Сброс с рольганга(брака) вперпед
	
	#S79_5 := "S79.5"; //Транспортер набора слоя ( брака) вперед
	#S79_6 := "S79.6"; //вилы( брака) вперед
	#E79_7 := "E79.7"; //вилы( брака) назад
	#S80_0 := "S80.0"; //опустить вилы ПФМ( брака)
	#E80_1 := "E80.1"; //поднять вилы ПФМ( брака)
	#S80_2 := "S80.2"; //Лифт ПФМ(брака) опустить
	#E80_3 := "E80.3"; //Лифт ПФМ(брака) поднять
	#S80_4 := "S80.4"; //поднять, опустить Подвижный борт(М235)
	#S80_5 := "S80.5"; //вперед подвижный борт(М235)
	#E80_6 := "E80.6"; //назад подвижный борт(М235)
	#S80_7 := "S80.7"; //0
	#Varalla106 := "Varalla106"; //резерв
	#Varalla107 := "Varalla107"; //резерв
	#Varalla108 := "Varalla108"; //резерв
	#Varalla109 := "Varalla109"; //резерв
	#Varalla110 := "Varalla110"; //резерв
	#Varalla111 := "Varalla111"; //резерв
	#Varalla112 := "Varalla112"; //резерв
	#Varalla113 := "Varalla113"; //резерв
	#S82_0 := "S82.0"; //Стоп ОР2
	#S81_1 := "S81.1"; //Приемный транспортер вперед ОР2
	#E82_2 := "E82.2"; //Приемный транспортер назад ОР2
	#S82_3 := "S82.3"; //Авто загрузка включена,выключена ОР2
	#S82_4 := "S82.4"; //Лифт загрузки поднять ОР2
	#E82_5 := "E82.5"; //Лифт загрузки опустить ОР2
	#S82_6 := "S82.6"; //Наклонный транспортер авто ОР2
	#E82_7 := "E82.7"; //Авто наклонный транспортер вперед ОР2
	#S83_0 := "S83.0"; //Ленточный транспортер удаления прокладок назад ОР2
	#E83_1 := "E83.1"; //Ленточный транспортер удаления прокладок вперед ОР2
	#E83_2 := "E83.2"; //Горка прокладок 1 авто ОР2
	#E83_3 := "E83.3"; //Горка прокладок 1 вперед ОР2(авто)
	#S83_4 := "S83.4"; //Квитирование зоны 1 ОР2
	#Varalla114 := "Varalla114"; //резерв
	#Varalla115 := "Varalla115"; //резерв
	#Varalla116 := "Varalla116"; //резерв
	#S84_0 := "S84.0"; //Стоп ОР3
	#S84_1 := "S84.1"; //Транспортер М317 прокладок вперед ОР3
	#E84_2 := "E84.2"; //Транспортер М317 прокладок назад ОР3
	#S84_3 := "S84.3"; //Дозировани включено ОР3
	#S84_4 := "S84.4"; //авто подача прокладок включена, выключена ОР3
	#S84_5 := "S84.5"; //Рейкоукладчик вниз ОР3
	#E84_6 := "E84.6"; //Рейкоукладчик вверх ОР3
	#S84_7 := "S84.7"; //Открыть стакан прокладки ОР3
	#E85_0 := "E85.0"; //Закрыть стакан прокладки ОР3
	#S85_1 := "S85.1"; //0
	#E85_2 := "E85.2"; //0
	#S85_3 := "S85.3"; //авто горка прокладок 2,3 ОР3
	#E85_4 := "E85.4"; //горка 2,3 прокладок вперед(авто) ОР3
	#S85_5 := "S85.5"; //М234 назад ОР3
	#E85_6 := "E85.6"; //М234 вперед транспортер прокладок перед крючками ОР3
	#S85_7 := "S85.7"; //Квитирование зоны прокладок ОР3
	#S86_0 := "S86.0"; //Лифт ПФМ вниз ОР3
	#E86_1 := "E86.1"; //ЛИфт ПФМ вверх ОР3
	#S86_2 := "S86.2"; //Ролики лифта ПФМ вперед ОР3
	#S86_3 := "S86.3"; //ПФМ Основное Авто включено, выключено ОР3
	#S86_4 := "S86.4"; //Подтверждение неисправности ОР3
	#S86_5 := "S86.5"; //датчик
	#Varalla117 := "Varalla117"; //резерв
	#Varalla118 := "Varalla118"; //резерв
	#S87_0 := "S87.0"; //Кнопка брака ОР1.1
	#S87_1 := "S87.1"; //Горка авто ОР1.1
	#E87_2 := "E87.2"; //Горка ОР1.1 (авто)
	#S87_3 := "S87.3"; //педаль 1ОР1.1
	#S87_4 := "S87.4"; //педаль2 ОР1.1
	#Varalla119 := "Varalla119"; //резерв
	#Varalla120 := "Varalla120"; //резерв
	#Varalla121 := "Varalla121"; //резерв
	#S88_0 := "S88.0"; //Стоп ОР4
	#K3_3 := "K3.3"; //работа подвижного борта ОР4
	#S88_2 := "S88.2"; //Выкатной транспортер 1 ПФМ назад ОР4
	#E88_3 := "E88.3"; //Выкатной транспортер 1 ПФМ вперед ОР4
	#S88_4 := "S88.4"; //Выкатной транспортер 2 ПФМ назад ОР4
	#S88_5 := "S88.5"; //Выкатной транспортер 2 ПФМ вперед ОР4
	#E88_6 := "E88.6"; //резерв ОР4
	#S88_7 := "S88.7"; //резерв ОР4
	#S89_0 := "S89.0"; //Выкатной транспортер 4 ПФМ назад ОР4
	#S89_1 := "S89.1"; //Выкатной транспортер 4 ПФМ вперед ОР4
	#S89_2 := "S89.2"; //Квитирование ОР4
	#S89_3 := "S89.3"; //датчик ОР4
	#Varalla122 := "Varalla122"; //резерв ОР4
	#Varalla123 := "Varalla123"; //резерв ОР4
	#Varalla124 := "Varalla124"; //резерв ОР4
	#Varalla125 := "Varalla125"; //резерв ОР4
	#S90_0 := "S90.0"; //Стоп ОР5
	#S90_1 := "S90.1"; //М331 вперед ленточный транспортер брака ОР5
	#S90_2 := "S90.2"; ; //М332 вперед сбрасыватель рольганга брака ОР5
	#Varalla126 := "Varalla126"; //резерв
	#S90_4 := "S90.4"; //Вилы ПФМ брака назад ОР5
	#E90_5 := "E90.5"; //Вилы ПФМ брака вперед ОР5
	#S90_6 := "S90.6"; //Опустить упоры формирования слоя на ПФМ брака ОР5
	#E90_7 := "E90.7"; //Поднять упоры формирования слоя на ПФМ брака ОР5
	#S91_0 := "S91.0"; //Лифт брака ПФМ опустить ОР5
	#E91_1 := "E91.1"; //Лифт брака ПФМ поднять ОР5
	#S91_2 := "S91.2"; //квитирование ПФМ 2
	#Varalla127 := "Varalla127"; //резерв
	#Varalla128 := "Varalla128"; //резерв
	#Varalla129 := "Varalla129"; //резерв
	#Varalla130 := "Varalla130"; //резерв
	#Varalla131 := "Varalla131"; //резерв
	#S214 := "234.4"; // пуск стоп приемного транспортера прокладок
	
	#btn_Drop_Defect(Sig:=#S87_0,
	                 set_Response_Time:=T#100ms);
	                 
	                 
	                 
	#btn_Cnrl_Mov_Side(Button_Sig:=#S80_4,
	                   set_Trembling_Time:=T#50ms,
	                   set_LongTapFixation_Time:=T#2s);
	
	#btn_Auto_Loading(Button_Sig:=#S76_5 OR #S82_3,
	                  set_Trembling_Time:=T#50ms
	);
	
	
	#btn_Auto_Sorting(Button_Sig:=#S77_5 OR #S86_3,
	                  set_Trembling_Time:=T#50ms
	);
	
	
	#btn_Auto_Gasket(Button_Sig:= #S79_1 OR #S84_4,
	                 set_Trembling_Time:=T#50ms
	);
	
	#btn_Auto_PFM_defective(Button_Sig:=#S79_3,
	                        set_Trembling_Time:=T#50ms
	);
	
	#btn_Reset_OP3(Button_Sig:="S86.4",
	               set_Trembling_Time:=T#50ms,
	               set_startLongTapFixation_Time:=T#1s,
	               set_LongTap_Time:=T#3s
	);
	
	
	#btn_Force_Finish(Sig := #S79_0,
	                  set_Response_Time := T#2s
	);
	
	
	#btn_ResetUporLine(Button_Sig:="S80.7",
	                   set_Trembling_Time:=T#50ms,
	                   set_LongTapFixation_Time:=T#2000ms);
	
	
	#"btn_Stop_M331/330"(Sig:="S90.1",
	                     set_Response_Time:=T#50ms);
	
	
	#btn_btnLenta_defect(Sig:="S90.2",
	                     set_Response_Time:=T#70ms);
	
END_FUNCTION_BLOCK

FUNCTION_BLOCK "Button_ShortTap"
{ S7_Optimized_Access := 'FALSE' }
VERSION : 0.1
   VAR_INPUT 
      Sig : Bool;
      set_Response_Time : Time;
   END_VAR

   VAR_OUTPUT 
      Out : Bool;
      fixed_tap : Bool;
   END_VAR

   VAR 
      Response_Timer {InstructionName := 'TON'; LibVersion := '1.0'; S7_SetPoint := 'False'} : TON;
   END_VAR


BEGIN
	#Out := FALSE;
	
	#Response_Timer(IN:=#Sig AND NOT #fixed_tap,
	                PT:=#set_Response_Time
	);
	
	#fixed_tap := (#fixed_tap OR #Response_Timer.Q) AND #Sig;
	
	#Out := #Response_Timer.Q;
END_FUNCTION_BLOCK

FUNCTION_BLOCK "ButtonSwitcher_PlusLongTap"
{ S7_Optimized_Access := 'FALSE' }
VERSION : 0.1
   VAR_INPUT 
      Button_Sig : Bool;   //  сигнал с кнопки
      set_Trembling_Time : Time;   //  время на дребезг контактов
      set_LongTapFixation_Time : Time;   //  время ожидания долгого тапа
   END_VAR

   VAR_OUTPUT 
      CMD_ON : Bool;   //  сигнал включения
      CMD_OFF : Bool;   //  сигнал выключения
      CMD_LongTap : Bool;   //  сигнал долго нажатия
   END_VAR

   VAR 
      Timer_LongTap_old : Bool;   //  сигнал с таймера на прошлой итерации
      inverter : Bool;   //  помогает инвертировать сигнал
      LongTap_Timer {InstructionName := 'TON'; LibVersion := '1.0'} : TON;   //  таймер долгого нажатия
   END_VAR


BEGIN
	#CMD_ON := FALSE;
	#CMD_OFF := FALSE;
	#CMD_LongTap := False;
	
	IF (#LongTap_Timer.ET > #set_Trembling_Time AND NOT #Button_Sig) THEN
	    #CMD_ON := NOT #inverter;
	    #CMD_OFF := #inverter;
	    #inverter := NOT #inverter;
	END_IF;
	
	#LongTap_Timer(IN := #Button_Sig,
	               PT := #set_LongTapFixation_Time
	);
	
	IF (#LongTap_Timer.Q AND NOT #Timer_LongTap_old) THEN
	    #CMD_LongTap := TRUE;
	END_IF;
	
	#Timer_LongTap_old := #LongTap_Timer.Q;
END_FUNCTION_BLOCK

FUNCTION_BLOCK "ButtonSwitcher"
{ S7_Optimized_Access := 'FALSE' }
VERSION : 0.1
   VAR_INPUT 
      Button_Sig : Bool;   //  сигнал с кнопки
      Reset_State : Bool;   // сброс состояния
      set_Trembling_Time : Time;   //  время на дребезг контактов
   END_VAR

   VAR_OUTPUT 
      CMD_ON : Bool;   //  сигнал включения
      CMD_OFF : Bool;   //  сигнал выключения
   END_VAR

   VAR 
      Timer_Sig_old : Bool;   //  сигнал с таймера на прошлой итерации
      inverter : Bool;   //  помогает инвертировать сигнал
      Trembling_Timer {InstructionName := 'TON'; LibVersion := '1.0'} : TON;   //  таймер на дребезг контактов
   END_VAR


BEGIN
	#CMD_ON :=  FALSE;
	#CMD_OFF := FALSE;
	
	#Trembling_Timer(IN := #Button_Sig,
	                 PT := #set_Trembling_Time
	);
	
	IF (#Reset_State) THEN
	    #inverter := FALSE;
	END_IF;
	
	IF #Trembling_Timer.Q AND NOT #Timer_Sig_old THEN
	    #CMD_ON := NOT #inverter;
	    #CMD_OFF := #inverter;
	    #inverter := NOT #inverter;
	END_IF;
	
	#Timer_Sig_old := #Trembling_Timer.Q;
END_FUNCTION_BLOCK

FUNCTION_BLOCK "ButtonShortLongTap"
{ S7_Optimized_Access := 'FALSE' }
VERSION : 0.1
   VAR_INPUT 
      Button_Sig : Bool;
      set_Trembling_Time : Time;
      set_startLongTapFixation_Time : Time;
      set_LongTap_Time : Time;
   END_VAR

   VAR_OUTPUT 
      ShortTap : Bool;   // короткий клик
      LongTap : Bool;   // длинное нажатие
      WaitingForLongTap : Bool;   // сигнал на лампочку кнопки
   END_VAR

   VAR 
      Button_Sig_old : Bool;
      ButtonTimer_old : Bool;
      noTremble : Bool;
      ButtonTimer {InstructionName := 'TON'; LibVersion := '1.0'; S7_SetPoint := 'False'} : TON;
   END_VAR


BEGIN
	#ShortTap := FALSE;
	#LongTap := False;
	
	#ButtonTimer(IN:=#Button_Sig,
	             PT:=#set_LongTap_Time);
	
	IF (#ButtonTimer.Q) THEN
	    #LongTap := TRUE;
	    #WaitingForLongTap := FALSE;
	ELSIF (#ButtonTimer.ET > #set_startLongTapFixation_Time) THEN
	    #noTremble := FALSE;
	    #WaitingForLongTap := TRUE;
	ELSIF (#ButtonTimer.ET > #set_Trembling_Time) THEN
	    #noTremble := TRUE;
	END_IF;
	
	IF (NOT #Button_Sig) THEN
	    #WaitingForLongTap := FALSE;
	    #ShortTap := #noTremble;
	    #noTremble := FALSE;
	END_IF;
	
	#ButtonTimer_old := #ButtonTimer.Q;
	#Button_Sig_old := #Button_Sig;
END_FUNCTION_BLOCK

FUNCTION_BLOCK "Button_PlusLongTap"
{ S7_Optimized_Access := 'FALSE' }
VERSION : 0.1
   VAR_INPUT 
      Button_Sig : Bool;   //  сигнал с кнопки
      set_Trembling_Time : Time;   //  время на дребезг контактов
      set_LongTapFixation_Time : Time;   //  время ожидания долгого тапа
   END_VAR

   VAR_OUTPUT 
      CMD_ON : Bool;   //  сигнал включения
      CMD_LongTap : Bool;   //  сигнал долго нажатия
   END_VAR

   VAR 
      Timer_LongTap_old : Bool;   //  сигнал с таймера на прошлой итерации
      LongTap_Timer {InstructionName := 'TON'; LibVersion := '1.0'} : TON;   //  таймер долгого нажатия
   END_VAR


BEGIN
	#CMD_ON := FALSE;
	#CMD_LongTap := False;
	
	IF (#LongTap_Timer.ET > #set_Trembling_Time AND NOT #Button_Sig) THEN
	    #CMD_ON := TRUE;
	END_IF;
	
	#LongTap_Timer(IN := #Button_Sig,
	               PT := #set_LongTapFixation_Time
	);
	
	IF (#LongTap_Timer.Q AND NOT #Timer_LongTap_old) THEN
	    #CMD_LongTap := TRUE;
	END_IF;
	
	#Timer_LongTap_old := #LongTap_Timer.Q;
END_FUNCTION_BLOCK

FUNCTION_BLOCK "Counter_1"   // FB20, LAD
AUTHOR : PSIfunc
VERSION : 0.1
// stored: AutoNumber true, IsIECCheckEnabled false, UDAEnableTagReadback false
   VAR
      SW_GATE_timer : TON;
   END_VAR
BEGIN

REGION Network 1
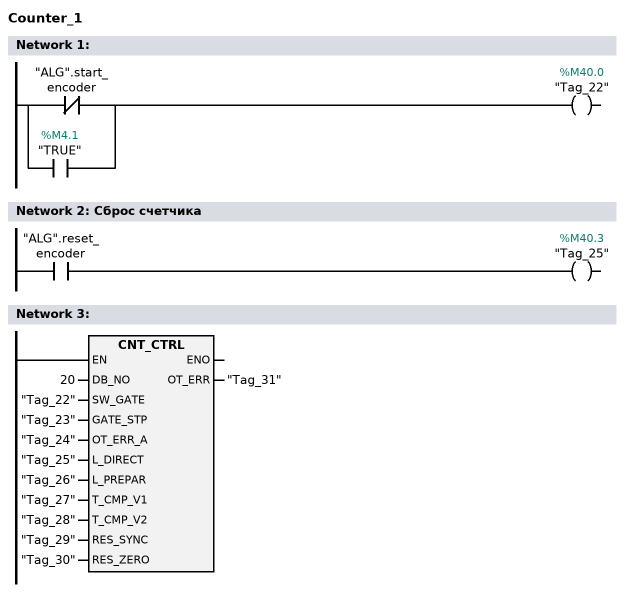
   RUNG wire#powerrail
      I_Contact( "ALG".start_encoder )
      wire#w1
      Coil( "Tag_22" )
   END_RUNG
   RUNG wire#powerrail
      Contact( "TRUE" )
   END_RUNG wire#w1
   // the same network as SCL:
   "Tag_22" := NOT "ALG".start_encoder OR "TRUE";
END_REGION

REGION Network 2: Сброс счетчика
   RUNG wire#powerrail
      Contact( "ALG".reset_encoder )
      Coil( "Tag_25" )
   END_RUNG
   // the same network as SCL:
   "Tag_25" := "ALG".reset_encoder;
END_REGION

REGION Network 3
   RUNG wire#powerrail
      CNT_CTRL(DB_NO := 20, SW_GATE := "Tag_22", GATE_STP := "Tag_23", OT_ERR_A := "Tag_24", L_DIRECT := "Tag_25", L_PREPAR := "Tag_26", T_CMP_V1 := "Tag_27", T_CMP_V2 := "Tag_28", RES_SYNC := "Tag_29", RES_ZERO := "Tag_30", OT_ERR => "Tag_31")
   END_RUNG
   // the same network as SCL:
   CNT_CTRL(DB_NO := 20,
            SW_GATE := "Tag_22",
            GATE_STP := "Tag_23",
            OT_ERR_A := "Tag_24",
            L_DIRECT := "Tag_25",
            L_PREPAR := "Tag_26",
            T_CMP_V1 := "Tag_27",
            T_CMP_V2 := "Tag_28",
            RES_SYNC := "Tag_29",
            RES_ZERO := "Tag_30",
            OT_ERR => "Tag_31");
END_REGION
END_FUNCTION_BLOCK

FUNCTION_BLOCK "Безопасность"   // FB1, LAD
VERSION : 0.1
// stored: AutoNumber true, IsIECCheckEnabled false, UDAEnableTagReadback false
   VAR DB_SPECIFIC
      Trig61 : Bool;
      Trig62 : Bool;
      Trig63 : Bool;
      Trig64 : Bool;
      Trig65 : Bool;
      Trig66 : Bool;
      Trig67 : Bool;
      Trig69 : Bool;
      Trig68 : Bool;
      ProhibitionLoading : Bool := true;
      ProhibitionDefect : Bool := true;
      ProhibitionSorting : Bool := true;
      ProhibitionGasket : Bool := true;
   END_VAR
   VAR_TEMP
      AlarmReset : Bool;
   END_VAR
   VAR_TEMP   // added for the SCL form of the ladder/FBD networks
      _w1 : Bool;
      _w2 : Bool;
      _s5time1 : S5Time;
   END_VAR
BEGIN

REGION Network 1: Реле безопастности К10 ОСНОВНАЯ напряжение управления
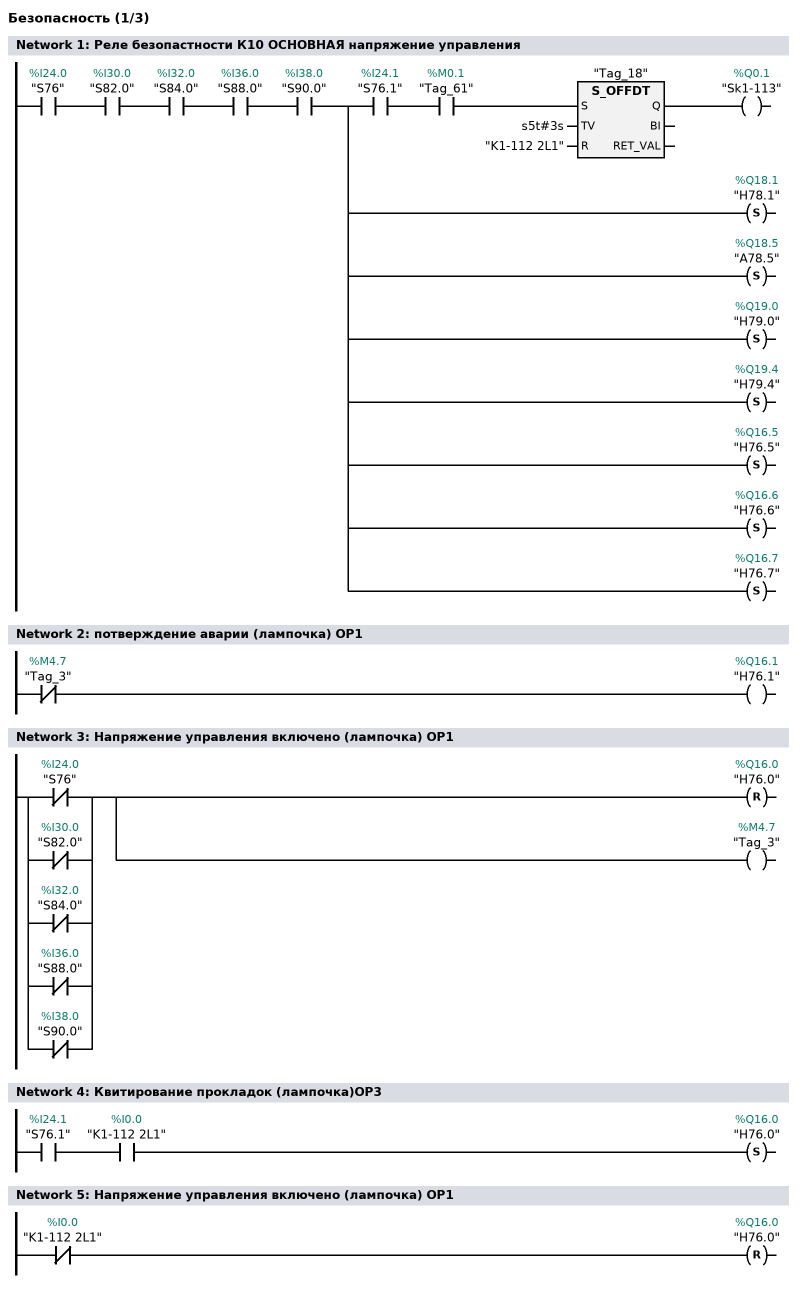
   RUNG wire#powerrail
      Contact( "S76" )
      Contact( "S82.0" )
      Contact( "S84.0" )
      Contact( "S88.0" )
      Contact( "S90.0" )
      wire#w1
      Contact( "S76.1" )
      Contact( "Tag_61" )
      S_OFFDT(T_NO := "Tag_18", TV := s5t#3s, R := "K1-112 2L1", BI =>, RET_VAL =>)
      Coil( "Sk1-113" )
   END_RUNG
   RUNG wire#w1
      S_Coil( "H78.1" )
   END_RUNG
   RUNG wire#w1
      S_Coil( "A78.5" )
   END_RUNG
   RUNG wire#w1
      S_Coil( "H79.0" )
   END_RUNG
   RUNG wire#w1
      S_Coil( "H79.4" )
   END_RUNG
   RUNG wire#w1
      S_Coil( "H76.5" )
   END_RUNG
   RUNG wire#w1
      S_Coil( "H76.6" )
   END_RUNG
   RUNG wire#w1
      S_Coil( "H76.7" )
   END_RUNG
   // the same network as SCL:
   #_w1 := "S76" AND "S82.0" AND "S84.0" AND "S88.0" AND "S90.0";
   #_s5time1 := S_OFFDT(T_NO := "Tag_18",
                        S := #_w1 AND "S76.1" AND "Tag_61",
                        TV := s5t#3s,
                        R := "K1-112 2L1",
                        Q => #_w2);
   "Sk1-113" := #_w2;
   IF #_w1 THEN
       "H78.1" := TRUE;
       "A78.5" := TRUE;
       "H79.0" := TRUE;
       "H79.4" := TRUE;
       "H76.5" := TRUE;
       "H76.6" := TRUE;
       "H76.7" := TRUE;
   END_IF;
END_REGION

REGION Network 2: потверждение аварии (лампочка) ОР1
   RUNG wire#powerrail
      I_Contact( "Tag_3" )
      Coil( "H76.1" )
   END_RUNG
   // the same network as SCL:
   "H76.1" := NOT "Tag_3";
END_REGION

REGION Network 3: Напряжение управления включено (лампочка) ОР1
   RUNG wire#powerrail
      I_Contact( "S76" )
      wire#w1
      R_Coil( "H76.0" )
   END_RUNG
   RUNG wire#powerrail
      I_Contact( "S82.0" )
   END_RUNG wire#w1
   RUNG wire#powerrail
      I_Contact( "S84.0" )
   END_RUNG wire#w1
   RUNG wire#powerrail
      I_Contact( "S88.0" )
   END_RUNG wire#w1
   RUNG wire#powerrail
      I_Contact( "S90.0" )
   END_RUNG wire#w1
   RUNG wire#w1
      Coil( "Tag_3" )
   END_RUNG
   // the same network as SCL:
   #_w1 := NOT "S76" OR NOT "S82.0" OR NOT "S84.0" OR NOT "S88.0" OR NOT "S90.0";
   IF #_w1 THEN "H76.0" := FALSE; END_IF;
   "Tag_3" := #_w1;
END_REGION

REGION Network 4: Квитирование прокладок (лампочка)ОР3
   RUNG wire#powerrail
      Contact( "S76.1" )
      Contact( "K1-112 2L1" )
      S_Coil( "H76.0" )
   END_RUNG
   // the same network as SCL:
   IF "S76.1" AND "K1-112 2L1" THEN "H76.0" := TRUE; END_IF;
END_REGION

REGION Network 5: Напряжение управления включено (лампочка) ОР1
   RUNG wire#powerrail
      I_Contact( "K1-112 2L1" )
      R_Coil( "H76.0" )
   END_RUNG
   // the same network as SCL:
   IF NOT "K1-112 2L1" THEN "H76.0" := FALSE; END_IF;
END_REGION

REGION Network 6: потверждение аварии (лампочка) ОР1
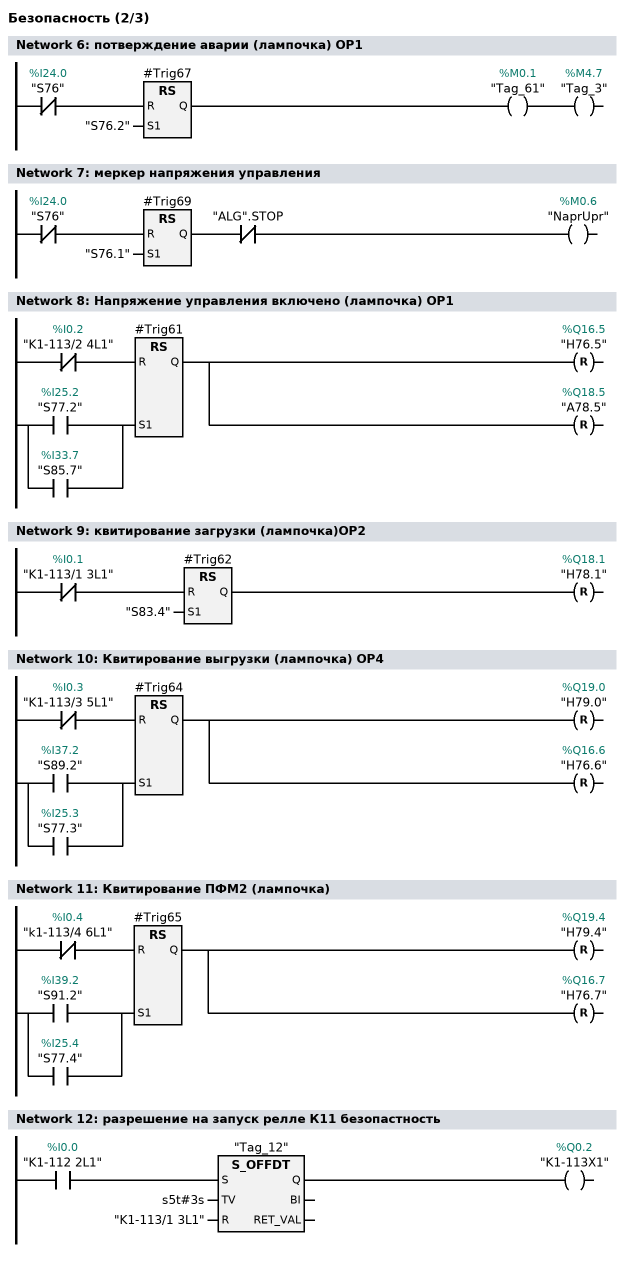
   RUNG wire#powerrail
      I_Contact( "S76" )
      S_RS(operand := #Trig67, s1 := "S76.2")
      Coil( "Tag_61" )
      Coil( "Tag_3" )
   END_RUNG
   // the same network as SCL:
   IF NOT "S76" THEN
       #Trig67 := FALSE;   // RS flip-flop
   END_IF;
   IF "S76.2" THEN #Trig67 := TRUE; END_IF;
   "Tag_61" := #Trig67;
   "Tag_3" := #Trig67;
END_REGION

REGION Network 7: меркер напряжения управления
   RUNG wire#powerrail
      I_Contact( "S76" )
      S_RS(operand := #Trig69, s1 := "S76.1")
      I_Contact( "ALG".STOP )
      Coil( "NaprUpr" )
   END_RUNG
   // the same network as SCL:
   IF NOT "S76" THEN
       #Trig69 := FALSE;   // RS flip-flop
   END_IF;
   IF "S76.1" THEN #Trig69 := TRUE; END_IF;
   "NaprUpr" := #Trig69 AND NOT "ALG".STOP;
END_REGION

REGION Network 8: Напряжение управления включено (лампочка) ОР1
   RUNG wire#powerrail
      I_Contact( "K1-113/2 4L1" )
      S_RS(operand := #Trig61, s1 := wire#w1)
      wire#w2
      R_Coil( "H76.5" )
   END_RUNG
   RUNG wire#powerrail
      Contact( "S77.2" )
   END_RUNG wire#w1
   RUNG wire#powerrail
      Contact( "S85.7" )
   END_RUNG wire#w1
   RUNG wire#w2
      R_Coil( "A78.5" )
   END_RUNG
   // the same network as SCL:
   IF NOT "K1-113/2 4L1" THEN
       #Trig61 := FALSE;   // RS flip-flop
   END_IF;
   IF "S77.2" OR "S85.7" THEN #Trig61 := TRUE; END_IF;
   IF #Trig61 THEN
       "H76.5" := FALSE;
       "A78.5" := FALSE;
   END_IF;
END_REGION

REGION Network 9: квитирование загрузки (лампочка)ОР2
   RUNG wire#powerrail
      I_Contact( "K1-113/1 3L1" )
      S_RS(operand := #Trig62, s1 := "S83.4")
      R_Coil( "H78.1" )
   END_RUNG
   // the same network as SCL:
   IF NOT "K1-113/1 3L1" THEN
       #Trig62 := FALSE;   // RS flip-flop
   END_IF;
   IF "S83.4" THEN #Trig62 := TRUE; END_IF;
   IF #Trig62 THEN "H78.1" := FALSE; END_IF;
END_REGION

REGION Network 10: Квитирование выгрузки (лампочка) ОР4
   RUNG wire#powerrail
      I_Contact( "K1-113/3 5L1" )
      S_RS(operand := #Trig64, s1 := wire#w1)
      wire#w2
      R_Coil( "H79.0" )
   END_RUNG
   RUNG wire#powerrail
      Contact( "S89.2" )
   END_RUNG wire#w1
   RUNG wire#powerrail
      Contact( "S77.3" )
   END_RUNG wire#w1
   RUNG wire#w2
      R_Coil( "H76.6" )
   END_RUNG
   // the same network as SCL:
   IF NOT "K1-113/3 5L1" THEN
       #Trig64 := FALSE;   // RS flip-flop
   END_IF;
   IF "S89.2" OR "S77.3" THEN #Trig64 := TRUE; END_IF;
   IF #Trig64 THEN
       "H79.0" := FALSE;
       "H76.6" := FALSE;
   END_IF;
END_REGION

REGION Network 11: Квитирование ПФМ2 (лампочка)
   RUNG wire#powerrail
      I_Contact( "k1-113/4 6L1" )
      S_RS(operand := #Trig65, s1 := wire#w1)
      wire#w2
      R_Coil( "H79.4" )
   END_RUNG
   RUNG wire#powerrail
      Contact( "S91.2" )
   END_RUNG wire#w1
   RUNG wire#powerrail
      Contact( "S77.4" )
   END_RUNG wire#w1
   RUNG wire#w2
      R_Coil( "H76.7" )
   END_RUNG
   // the same network as SCL:
   IF NOT "k1-113/4 6L1" THEN
       #Trig65 := FALSE;   // RS flip-flop
   END_IF;
   IF "S91.2" OR "S77.4" THEN #Trig65 := TRUE; END_IF;
   IF #Trig65 THEN
       "H79.4" := FALSE;
       "H76.7" := FALSE;
   END_IF;
END_REGION

REGION Network 12: разрешение на запуск релле К11 безопастность
   RUNG wire#powerrail
      Contact( "K1-112 2L1" )
      S_OFFDT(T_NO := "Tag_12", TV := s5t#3s, R := "K1-113/1 3L1", BI =>, RET_VAL =>)
      Coil( "K1-113X1" )
   END_RUNG
   // the same network as SCL:
   #_s5time1 := S_OFFDT(T_NO := "Tag_12", S := "K1-112 2L1", TV := s5t#3s, R := "K1-113/1 3L1", Q => #_w1);
   "K1-113X1" := #_w1;
END_REGION

